# B&R Automation Studio project NAELD004C00R10L518F00 (part 17)

#### Act_OptP1025Save.st
```iecst
ACTION Act_OptP1025Save:

	IF tyP1025McSetAIVComm.tyAIVComm.tyNumSvrPort.bRtCompl OR tyP1025McSetAIVComm.tyAIVComm.tyNumAllwClntPort.bRtCompl
		OR tyP1025McSetAIVComm.tyAIVComm.tyStringAllwClntIP.bRtCompl THEN

		fUIInRtStatHide(ADR(tyCommon.tySet.tyBtnSave.uiMaskRtStat));

		 tyP1025McSetAIVComm.tyAIVComm.tyNumSvrPort.bRtCompl		:= FALSE;
		 tyP1025McSetAIVComm.tyAIVComm.tyNumAllwClntPort.bRtCompl	:= FALSE;
	 	 tyP1025McSetAIVComm.tyAIVComm.tyStringAllwClntIP.bRtCompl	:= FALSE;

	END_IF

	IF tyCommon.tySet.tyBtnSave.bRtCompl = TRUE THEN

		IF usiSaveAIVCommStep = 0 THEN
			//Verify IP Address Valid
			IF tyP1025McSetAIVComm.tyAIVComm.tyStringAllwClntIP.sValue <> '' THEN

				IF fIPValid(tyP1025McSetAIVComm.tyAIVComm.tyStringAllwClntIP.sValue, ADR(a_iIPPart1)) = TRUE THEN
					usiSaveAIVCommStep	:= 1;
				ELSE
					usiSaveAIVCommStep	:= 99;
				END_IF

			ELSE
				usiSaveAIVCommStep	:= 1;
			END_IF

		ELSIF usiSaveAIVCommStep = 1 THEN
			//Save Param
			tyMcParamWr.tyAIVComm.uiSvrPort			:=  DINT_TO_UINT(tyP1025McSetAIVComm.tyAIVComm.tyNumSvrPort.diValue);
			tyMcParamWr.tyAIVComm.uiClientPort		:=  DINT_TO_UINT(tyP1025McSetAIVComm.tyAIVComm.tyNumAllwClntPort.diValue);
			tyMcParamWr.tyAIVComm.sClientAddress	:=  tyP1025McSetAIVComm.tyAIVComm.tyStringAllwClntIP.sValue;

			eMcParamAct	:= McParamActWrite;

			IF p_eMcParamStat = McParamActWrite AND p_eMcParamStatus = Done THEN

				eMcParamAct	:= McParamActIdle;

				//Update BackUp Param
				tyP1025McSetAIVComm.tyAIVCommBkUp	:= tyP1025McSetAIVComm.tyAIVComm;

				//Reconnect
				bAIVCommReconnect	:= TRUE;

				usiSaveAIVCommStep	:= 2;

			ELSIF p_eMcParamStatus = Error THEN

				p_tyC0008MsgBox ACCESS ADR(tyP1025McSetAIVComm.tyMsgBoxSaveErr);

				IF tyP1025McSetAIVComm.tyMsgBoxSaveErr.tyBtnNo.bRtCompl = TRUE THEN
					tyP1025McSetAIVComm.tyMsgBoxSaveErr.tyBtnNo.bRtCompl	:= FALSE;
					tyP1025McSetAIVComm.tyMsgBoxSaveErr.tyBtnNo.bValue		:= FALSE;

					p_tyC0008MsgBox ACCESS ADR(tyP1025McSetAIVComm.tyMsgBoxHide);

					//Restore Param
					tyP1025McSetAIVComm.tyAIVComm	:= tyP1025McSetAIVComm.tyAIVCommBkUp;
					tyMcParamWr						:= p_tyMcParamCurr;

					tyCommon.tySet.tyBtnSave.bRtCompl	:= FALSE;
					fUIInRtStatOff(ADR(tyCommon.tySet.tyBtnSave.uiMaskRtStat));
				END_IF

			END_IF

		ELSIF usiSaveAIVCommStep = 2 THEN
			//Done
			bAIVCommReconnect	:= FALSE;

			usiSaveAIVCommStep	:= 0;

			tyCommon.tySet.tyBtnSave.bRtCompl 	:= FALSE;
			fUIInRtStatOff(ADR(tyCommon.tySet.tyBtnSave.uiMaskRtStat));

		ELSIF usiSaveAIVCommStep = 99 THEN
			//Message: IP Address Invalid
			p_tyC0008MsgBox ACCESS ADR(tyP1025McSetAIVComm.tyMsgBoxIPAddrInvalid);

			IF tyP1025McSetAIVComm.tyMsgBoxIPAddrInvalid.tyBtnNo.bRtCompl = TRUE THEN
				tyP1025McSetAIVComm.tyMsgBoxIPAddrInvalid.tyBtnNo.bRtCompl	:= FALSE;
				tyP1025McSetAIVComm.tyMsgBoxIPAddrInvalid.tyBtnNo.bValue	:= FALSE;

				p_tyC0008MsgBox ACCESS ADR(tyP1025McSetAIVComm.tyMsgBoxHide);

				//Restore Param
				tyP1025McSetAIVComm.tyAIVComm	:= tyP1025McSetAIVComm.tyAIVCommBkUp;

				usiSaveAIVCommStep	:= 0;

				tyCommon.tySet.tyBtnSave.bRtCompl	:= FALSE;
				fUIInRtStatOff(ADR(tyCommon.tySet.tyBtnSave.uiMaskRtStat));
			END_IF

		END_IF

	END_IF

END_ACTION
```

#### Act_EntP1026Disp.st
```iecst
ACTION Act_EntP1026Disp:

	//Access Address
	p_tyC0002FullMask ACCESS ADR(tyP1026McSetTeach.tyFullMaskHide);

	p_tyC0004Navi ACCESS ADR(tyP1026McSetTeach.tyNaviBack);

	p_tyC0005Main ACCESS ADR(tyCommon.tyMain);

	p_tyC0007Notif ACCESS ADR(tyCommon.tyNotif);

	p_tyC0008MsgBox ACCESS ADR(tyP1026McSetTeach.tyMsgBoxHide);

	p_tyC0009Info ACCESS ADR(tyCommon.tyInfo);

	p_tyP1026InOutletShutterFB ACCESS ADR(tyP1026McSetTeach.tyInOutletShutterFB);

	IF bTeachTravPosA = TRUE THEN
		p_tyP1026McSetTeach ACCESS ADR(tyP1026McSetTeach.tyTeachTravPosA);
		p_tyC0001MotionStd ACCESS ADR(tyP1026McSetTeach.tyMotionStdTrav);

	ELSIF bTeachTravPosB = TRUE THEN
		p_tyP1026McSetTeach ACCESS ADR(tyP1026McSetTeach.tyTeachTravPosB);
		p_tyC0001MotionStd ACCESS ADR(tyP1026McSetTeach.tyMotionStdTrav);

	ELSIF bTeachLifterPosA = TRUE THEN
		p_tyP1026McSetTeach ACCESS ADR(tyP1026McSetTeach.tyTeachLifterPosA);
		p_tyC0001MotionStd ACCESS ADR(tyP1026McSetTeach.tyMotionStdLifter);

	ELSIF bTeachLifterPosB = TRUE THEN
		p_tyP1026McSetTeach ACCESS ADR(tyP1026McSetTeach.tyTeachLifterPosB);
		p_tyC0001MotionStd ACCESS ADR(tyP1026McSetTeach.tyMotionStdLifter);

	END_IF

	//Display
	//Traverser
	tyP1026McSetTeach.tyMotionStdTrav.tyBtnPwr.bValue	:= p_bTravPwrOn;

	//Lifter
	tyP1026McSetTeach.tyMotionStdLifter.tyBtnPwr.bValue	:= p_bLifterBtmPwrOn;

//	bTeachServo		:= TRUE;
END_ACTION
```

#### Act_ExitP1026.st
```iecst
ACTION Act_ExitP1026:

	usiChgPage	:= 1;

	//Manual Deactivated
	bManualMod	:= FALSE;

	//Reset UI
	bJogSlow				:= FALSE;
	bJogFast				:= FALSE;
	fbJogSlowToFastDlyTm.IN	:= FALSE;

	fbLmtRstTm(IN := FALSE);
	//bypass curtain sensor
	bBypCurtainSen := FALSE;
	bBypCurtainPBLED := FALSE;
	tyP1026McSetTeach.tyTeachTravPosA.tyBtn4.bValue				:= FALSE;
	tyP1026McSetTeach.tyTeachTravPosB.tyBtn4.bValue				:= FALSE;
	tyP1026McSetTeach.tyTeachLifterPosA.tyBtn4.bValue				:= FALSE;
	tyP1026McSetTeach.tyTeachLifterPosB.tyBtn4.bValue				:= FALSE;

	//Traverser
	tyP1026McSetTeach.tyMotionStdTrav.tyBtnPwr.bRtCompl				:= FALSE;
	tyP1026McSetTeach.tyMotionStdTrav.tyBtnStop.bRtCompl			:= FALSE;
	tyP1026McSetTeach.tyMotionStdTrav.tyBtnOrigin.bRtCompl			:= FALSE;
	tyP1026McSetTeach.tyMotionStdTrav.tyBtnRst.bRtCompl				:= FALSE;
	tyP1026McSetTeach.tyMotionStdTrav.tyBtnMovAbs.bRtCompl			:= FALSE;
	tyP1026McSetTeach.tyMotionStdTrav.tyBtnMovRel.bRtCompl			:= FALSE;
	tyP1026McSetTeach.tyMotionStdTrav.tyBtnJogFront.bRtCompl		:= FALSE;
	tyP1026McSetTeach.tyMotionStdTrav.tyBtnJogRear.bRtCompl			:= FALSE;

	tyP1026McSetTeach.tyTeachTravPosA.tyBtn2.bRtCompl				:= FALSE;
	tyP1026McSetTeach.tyTeachTravPosB.tyBtn2.bRtCompl				:= FALSE;

	tyP1026McSetTeach.tyMotionStdTrav.tyBtnPwr.bValue				:= FALSE;
	tyP1026McSetTeach.tyMotionStdTrav.tyBtnStop.bValue				:= TRUE;
	tyP1026McSetTeach.tyMotionStdTrav.tyBtnOrigin.bValue			:= FALSE;
	tyP1026McSetTeach.tyMotionStdTrav.tyBtnRst.bValue				:= FALSE;
	tyP1026McSetTeach.tyMotionStdTrav.tyBtnMovAbs.bValue			:= FALSE;
	tyP1026McSetTeach.tyMotionStdTrav.tyBtnMovRel.bValue			:= FALSE;
	tyP1026McSetTeach.tyMotionStdTrav.tyBtnJogFront.bValue			:= FALSE;
	tyP1026McSetTeach.tyMotionStdTrav.tyBtnJogRear.bValue			:= FALSE;

	tyP1026McSetTeach.tyTeachTravPosA.tyBtn2.bValue					:= FALSE;
	tyP1026McSetTeach.tyTeachTravPosB.tyBtn2.bValue					:= FALSE;

	tyP1026McSetTeach.tyMotionStdTrav.tyBtnPwr.bRtLk				:= FALSE;
	tyP1026McSetTeach.tyMotionStdTrav.tyBtnStop.bRtLk				:= TRUE;
	tyP1026McSetTeach.tyMotionStdTrav.tyBtnOrigin.bRtLk				:= FALSE;
	tyP1026McSetTeach.tyMotionStdTrav.tyBtnRst.bRtLk				:= FALSE;
	tyP1026McSetTeach.tyMotionStdTrav.tyBtnMovAbs.bRtLk				:= FALSE;
	tyP1026McSetTeach.tyMotionStdTrav.tyBtnMovRel.bRtLk				:= FALSE;
	tyP1026McSetTeach.tyMotionStdTrav.tyBtnJogFront.bRtLk			:= FALSE;
	tyP1026McSetTeach.tyMotionStdTrav.tyBtnJogRear.bRtLk			:= FALSE;

	tyP1026McSetTeach.tyTeachTravPosA.tyBtn2.bRtLk					:= FALSE;
	tyP1026McSetTeach.tyTeachTravPosB.tyBtn2.bRtLk					:= FALSE;

	tyP1026McSetTeach.tyMotionStdTrav.tyBtnPwr.uiMaskRtStat			:= TRUE;
	tyP1026McSetTeach.tyMotionStdTrav.tyBtnOrigin.uiMaskRtStat		:= FALSE;
	tyP1026McSetTeach.tyMotionStdTrav.tyBtnRst.uiMaskRtStat			:= TRUE;
	tyP1026McSetTeach.tyMotionStdTrav.tyBtnMovAbs.uiMaskRtStat		:= FALSE;
	tyP1026McSetTeach.tyMotionStdTrav.tyBtnMovRel.uiMaskRtStat		:= FALSE;
	tyP1026McSetTeach.tyMotionStdTrav.tyBtnJogFront.uiMaskRtStat	:= FALSE;
	tyP1026McSetTeach.tyMotionStdTrav.tyBtnJogRear.uiMaskRtStat		:= FALSE;

	tyP1026McSetTeach.tyTeachTravPosA.tyBtn2.uiMaskRtStat			:= FALSE;
	tyP1026McSetTeach.tyTeachTravPosB.tyBtn2.uiMaskRtStat			:= FALSE;

	//Lifter
	tyP1026McSetTeach.tyMotionStdLifter.tyBtnPwr.bRtCompl			:= FALSE;
	tyP1026McSetTeach.tyMotionStdLifter.tyBtnStop.bRtCompl			:= FALSE;
	tyP1026McSetTeach.tyMotionStdLifter.tyBtnOrigin.bRtCompl		:= FALSE;
	tyP1026McSetTeach.tyMotionStdLifter.tyBtnRst.bRtCompl			:= FALSE;
	tyP1026McSetTeach.tyMotionStdLifter.tyBtnMovAbs.bRtCompl		:= FALSE;
	tyP1026McSetTeach.tyMotionStdLifter.tyBtnMovRel.bRtCompl		:= FALSE;
	tyP1026McSetTeach.tyMotionStdLifter.tyBtnJogUp.bRtCompl			:= FALSE;
	tyP1026McSetTeach.tyMotionStdLifter.tyBtnJogDown.bRtCompl		:= FALSE;

	tyP1026McSetTeach.tyTeachLifterPosA.tyBtn2.bRtCompl				:= FALSE;
	tyP1026McSetTeach.tyTeachLifterPosB.tyBtn2.bRtCompl				:= FALSE;

	tyP1026McSetTeach.tyMotionStdLifter.tyBtnPwr.bValue				:= FALSE;
	tyP1026McSetTeach.tyMotionStdLifter.tyBtnStop.bValue			:= TRUE;
	tyP1026McSetTeach.tyMotionStdLifter.tyBtnOrigin.bValue			:= FALSE;
	tyP1026McSetTeach.tyMotionStdLifter.tyBtnRst.bValue				:= FALSE;
	tyP1026McSetTeach.tyMotionStdLifter.tyBtnMovAbs.bValue			:= FALSE;
	tyP1026McSetTeach.tyMotionStdLifter.tyBtnMovRel.bValue			:= FALSE;
	tyP1026McSetTeach.tyMotionStdLifter.tyBtnJogUp.bValue			:= FALSE;
	tyP1026McSetTeach.tyMotionStdLifter.tyBtnJogDown.bValue			:= FALSE;

	tyP1026McSetTeach.tyTeachLifterPosA.tyBtn2.bValue				:= FALSE;
	tyP1026McSetTeach.tyTeachLifterPosB.tyBtn2.bValue				:= FALSE;

	tyP1026McSetTeach.tyMotionStdLifter.tyBtnPwr.bRtLk				:= FALSE;
	tyP1026McSetTeach.tyMotionStdLifter.tyBtnStop.bRtLk				:= TRUE;
	tyP1026McSetTeach.tyMotionStdLifter.tyBtnOrigin.bRtLk			:= FALSE;
	tyP1026McSetTeach.tyMotionStdLifter.tyBtnRst.bRtLk				:= FALSE;
	tyP1026McSetTeach.tyMotionStdLifter.tyBtnMovAbs.bRtLk			:= FALSE;
	tyP1026McSetTeach.tyMotionStdLifter.tyBtnMovRel.bRtLk			:= FALSE;
	tyP1026McSetTeach.tyMotionStdLifter.tyBtnJogUp.bRtLk			:= FALSE;
	tyP1026McSetTeach.tyMotionStdLifter.tyBtnJogDown.bRtLk			:= FALSE;

	tyP1026McSetTeach.tyTeachLifterPosA.tyBtn2.bRtLk				:= FALSE;
	tyP1026McSetTeach.tyTeachLifterPosB.tyBtn2.bRtLk				:= FALSE;

	tyP1026McSetTeach.tyMotionStdLifter.tyBtnPwr.uiMaskRtStat		:= TRUE;
	tyP1026McSetTeach.tyMotionStdLifter.tyBtnOrigin.uiMaskRtStat	:= FALSE;
	tyP1026McSetTeach.tyMotionStdLifter.tyBtnRst.uiMaskRtStat		:= TRUE;
	tyP1026McSetTeach.tyMotionStdLifter.tyBtnMovAbs.uiMaskRtStat	:= FALSE;
	tyP1026McSetTeach.tyMotionStdLifter.tyBtnMovRel.uiMaskRtStat	:= FALSE;
	tyP1026McSetTeach.tyMotionStdLifter.tyBtnJogUp.uiMaskRtStat		:= FALSE;
	tyP1026McSetTeach.tyMotionStdLifter.tyBtnJogDown.uiMaskRtStat	:= FALSE;

	tyP1026McSetTeach.tyTeachLifterPosA.tyBtn2.uiMaskRtStat			:= FALSE;
	tyP1026McSetTeach.tyTeachLifterPosB.tyBtn2.uiMaskRtStat			:= FALSE;

END_ACTION
```

#### Act_OptP1026TravTeach.st
```iecst
ACTION Act_OptP1026TravTeach:

	IF tyP1026McSetTeach.tyTeachTravPosA.tyBtn1.bRtCompl = TRUE THEN

		p_tyC0008MsgBox ACCESS ADR(tyP1026McSetTeach.tyMsgBoxUpdtTravPosA);

		IF tyP1026McSetTeach.tyMsgBoxUpdtTravPosA.tyBtnNo.bRtCompl THEN
			tyP1026McSetTeach.tyMsgBoxUpdtTravPosA.tyBtnNo.bRtCompl	:= FALSE;
			tyP1026McSetTeach.tyMsgBoxUpdtTravPosA.tyBtnNo.bValue	:= FALSE;

			p_tyC0008MsgBox ACCESS ADR(tyP1026McSetTeach.tyMsgBoxHide);

			//Write Actual Position To Machine Settings
			tyP1021McSetGen.tyGen.tyNumTravPosLaneA.diValue 	:= p_diTravActualPos;
			tyP1021McSetGen.tyGen.tyNumTravPosLaneA.bRtCompl	:= TRUE;

			//Back To Machine Settings
			eChgPage	:= UIP1021McSetGen;

			fUIInRtStatHide(ADR(tyCommon.tySet.tyBtnSave.uiMaskRtStat));

			tyP1026McSetTeach.tyTeachTravPosA.tyBtn1.bRtCompl	:= FALSE;
			tyP1026McSetTeach.tyTeachTravPosA.tyBtn1.bValue		:= FALSE;

		END_IF

	ELSIF tyP1026McSetTeach.tyTeachTravPosB.tyBtn1.bRtCompl = TRUE THEN

		p_tyC0008MsgBox ACCESS ADR(tyP1026McSetTeach.tyMsgBoxUpdtTravPosB);

		IF tyP1026McSetTeach.tyMsgBoxUpdtTravPosB.tyBtnNo.bRtCompl THEN
			tyP1026McSetTeach.tyMsgBoxUpdtTravPosB.tyBtnNo.bRtCompl := FALSE;
			tyP1026McSetTeach.tyMsgBoxUpdtTravPosB.tyBtnNo.bValue 	:= FALSE;

			p_tyC0008MsgBox ACCESS ADR(tyP1026McSetTeach.tyMsgBoxHide);

			//Write Actual Position To Machine Settings
			tyP1021McSetGen.tyGen.tyNumTravPosLaneB.diValue 	:= p_diTravActualPos;
			tyP1021McSetGen.tyGen.tyNumTravPosLaneB.bRtCompl	:= TRUE;

			//Back To Machine Settings
			eChgPage	:= UIP1021McSetGen;

			fUIInRtStatHide(ADR(tyCommon.tySet.tyBtnSave.uiMaskRtStat));

			tyP1026McSetTeach.tyTeachTravPosB.tyBtn1.bRtCompl	:= FALSE;
			tyP1026McSetTeach.tyTeachTravPosB.tyBtn1.bValue		:= FALSE;

		END_IF

	END_IF

END_ACTION
```

#### Act_OptP1026TravFBCtrl.st
```iecst
ACTION Act_OptP1026TravFBCtrl:

	fbJogSlowToFastDlyTm.PT			:= T#2s;
	fbJogSlowToFastDlyTm;
	fbLmtRstTm;

//	IF EDGEPOS((p_udiTravAxisErrID = 21570 OR p_udiTravAxisErrID = 21571)
	IF EDGEPOS((p_bTravFwdLmtSen OR p_bTravRevLmtSen OR p_udiTravAxisErrID = 21570 OR p_udiTravAxisErrID = 21571)
		AND tyP1026McSetTeach.tyMotionStdTrav.tyBtnJogRear.bValue = FALSE
		AND tyP1026McSetTeach.tyMotionStdTrav.tyBtnJogFront.bValue = FALSE) THEN

		fbLmtRstTm.IN				:= TRUE;
	END_IF

	IF fbLmtRstTm.Q = TRUE THEN
		tyP1026McSetTeach.tyMotionStdTrav.tyBtnRst.bRtCompl		:= TRUE;
	END_IF

	IF (tyP1026McSetTeach.tyMotionStdTrav.tyBtnJogFront.bValue = FALSE AND tyP1026McSetTeach.tyMotionStdTrav.tyBtnJogRear.bValue = FALSE) AND (p_bTravJogging = TRUE) THEN
		bJogStopTrav	:= TRUE;
	END_IF

	IF tyP1026McSetTeach.tyMotionStdTrav.tyBtnStop.bRtCompl = TRUE THEN
		eTravAct		:= TravActStop;

		IF p_eTravStat = TravActStop AND p_eTravStatus = Done THEN
			eTravAct	:= TravActIdle;

			tyP1026McSetTeach.tyMotionStdTrav.tyBtnStop.bRtCompl		:= FALSE;
			tyP1026McSetTeach.tyMotionStdTrav.tyBtnJogRear.bRtCompl		:= FALSE;
			tyP1026McSetTeach.tyMotionStdTrav.tyBtnJogFront.bRtCompl	:= FALSE;
			tyP1026McSetTeach.tyMotionStdTrav.tyBtnOrigin.bRtCompl		:= FALSE;
			tyP1026McSetTeach.tyMotionStdTrav.tyBtnMovAbs.bRtCompl		:= FALSE;
			tyP1026McSetTeach.tyMotionStdTrav.tyBtnMovRel.bRtCompl		:= FALSE;

			tyP1026McSetTeach.tyTeachTravPosA.tyBtn2.bRtCompl			:= FALSE;
			tyP1026McSetTeach.tyTeachTravPosB.tyBtn2.bRtCompl			:= FALSE;

			tyP1026McSetTeach.tyMotionStdTrav.tyBtnStop.bValue			:= TRUE;
			tyP1026McSetTeach.tyMotionStdTrav.tyBtnJogRear.bValue		:= FALSE;
			tyP1026McSetTeach.tyMotionStdTrav.tyBtnJogFront.bValue		:= FALSE;
			tyP1026McSetTeach.tyMotionStdTrav.tyBtnOrigin.bValue		:= FALSE;
			tyP1026McSetTeach.tyMotionStdTrav.tyBtnMovAbs.bValue		:= FALSE;
			tyP1026McSetTeach.tyMotionStdTrav.tyBtnMovRel.bValue		:= FALSE;
			tyP1026McSetTeach.tyTeachTravPosA.tyBtn2.bValue				:= FALSE;
			tyP1026McSetTeach.tyTeachTravPosB.tyBtn2.bValue				:= FALSE;

			tyP1026McSetTeach.tyMotionStdTrav.tyBtnStop.bRtLk			:= TRUE;
			tyP1026McSetTeach.tyMotionStdTrav.tyBtnJogRear.bRtLk		:= FALSE;
			tyP1026McSetTeach.tyMotionStdTrav.tyBtnJogFront.bRtLk		:= FALSE;
			tyP1026McSetTeach.tyMotionStdTrav.tyBtnOrigin.bRtLk			:= FALSE;
			tyP1026McSetTeach.tyMotionStdTrav.tyBtnMovAbs.bRtLk			:= FALSE;
			tyP1026McSetTeach.tyMotionStdTrav.tyBtnMovRel.bRtLk			:= FALSE;

			tyP1026McSetTeach.tyTeachTravPosA.tyBtn2.bRtLk						:= FALSE;
			tyP1026McSetTeach.tyTeachTravPosB.tyBtn2.bRtLk						:= FALSE;
		END_IF

	ELSIF (tyP1026McSetTeach.tyMotionStdTrav.tyBtnJogRear.bRtCompl = TRUE) OR (tyP1026McSetTeach.tyMotionStdTrav.tyBtnJogFront.bRtCompl = TRUE) OR (bJogStopTrav = TRUE) THEN
		bJogSlow					:= FALSE;
		bJogFast					:= FALSE;
		fbJogSlowToFastDlyTm.IN		:= FALSE;

		eTravAct		:= TravActJogStop;

		IF p_eTravStat = TravActJogStop AND p_eTravStatus = Done THEN
			eTravAct		:= TravActIdle;

			bJogStopTrav	:= FALSE;

			tyP1026McSetTeach.tyMotionStdTrav.tyBtnStop.bRtCompl		:= FALSE;
			tyP1026McSetTeach.tyMotionStdTrav.tyBtnJogRear.bRtCompl		:= FALSE;
			tyP1026McSetTeach.tyMotionStdTrav.tyBtnJogFront.bRtCompl	:= FALSE;
			tyP1026McSetTeach.tyMotionStdTrav.tyBtnOrigin.bRtCompl		:= FALSE;
			tyP1026McSetTeach.tyMotionStdTrav.tyBtnMovAbs.bRtCompl		:= FALSE;
			tyP1026McSetTeach.tyMotionStdTrav.tyBtnMovRel.bRtCompl		:= FALSE;
			tyP1026McSetTeach.tyTeachTravPosA.tyBtn2.bRtCompl			:= FALSE;
			tyP1026McSetTeach.tyTeachTravPosB.tyBtn2.bRtCompl			:= FALSE;

			tyP1026McSetTeach.tyMotionStdTrav.tyBtnStop.bValue			:= TRUE;
			tyP1026McSetTeach.tyMotionStdTrav.tyBtnJogRear.bValue		:= FALSE;
			tyP1026McSetTeach.tyMotionStdTrav.tyBtnJogFront.bValue		:= FALSE;
			tyP1026McSetTeach.tyMotionStdTrav.tyBtnOrigin.bValue		:= FALSE;
			tyP1026McSetTeach.tyMotionStdTrav.tyBtnMovAbs.bValue		:= FALSE;
			tyP1026McSetTeach.tyMotionStdTrav.tyBtnMovRel.bValue		:= FALSE;
			tyP1026McSetTeach.tyTeachTravPosA.tyBtn2.bValue				:= FALSE;
			tyP1026McSetTeach.tyTeachTravPosB.tyBtn2.bValue				:= FALSE;

			tyP1026McSetTeach.tyMotionStdTrav.tyBtnStop.bRtLk			:= TRUE;
			tyP1026McSetTeach.tyMotionStdTrav.tyBtnJogRear.bRtLk		:= FALSE;
			tyP1026McSetTeach.tyMotionStdTrav.tyBtnJogFront.bRtLk		:= FALSE;
			tyP1026McSetTeach.tyMotionStdTrav.tyBtnOrigin.bRtLk			:= FALSE;
			tyP1026McSetTeach.tyMotionStdTrav.tyBtnMovAbs.bRtLk			:= FALSE;
			tyP1026McSetTeach.tyMotionStdTrav.tyBtnMovRel.bRtLk			:= FALSE;
			tyP1026McSetTeach.tyTeachTravPosA.tyBtn2.bRtLk				:= FALSE;
			tyP1026McSetTeach.tyTeachTravPosB.tyBtn2.bRtLk				:= FALSE;
		END_IF

	ELSIF tyP1026McSetTeach.tyMotionStdTrav.tyBtnPwr.bRtCompl = TRUE THEN
		tyP1026McSetTeach.tyMotionStdTrav.tyBtnPwr.bRtLk				:= TRUE;

		IF tyP1026McSetTeach.tyMotionStdTrav.tyBtnPwr.bValue = TRUE THEN
			eTravAct		:= TravActPwrOn;

			IF p_eTravStat = TravActPwrOn AND p_eTravStatus = Done THEN
				eTravAct	:= TravActIdle;

				tyP1026McSetTeach.tyMotionStdTrav.tyBtnPwr.bRtCompl		:= FALSE;
				tyP1026McSetTeach.tyMotionStdTrav.tyBtnPwr.bRtLk		:= FALSE;
			END_IF
		ELSE
			eTravAct		:= TravActPwrOff;

			IF p_eTravStat = TravActPwrOff AND p_eTravStatus = Done THEN
				eTravAct	:= TravActIdle;

				tyP1026McSetTeach.tyMotionStdTrav.tyBtnPwr.bRtCompl		:= FALSE;
				tyP1026McSetTeach.tyMotionStdTrav.tyBtnPwr.bRtLk		:= FALSE;
			END_IF
		END_IF

	ELSIF tyP1026McSetTeach.tyMotionStdTrav.tyBtnOrigin.bRtCompl = TRUE THEN
		tyP1026McSetTeach.tyMotionStdTrav.tyBtnOrigin.bValue			:= TRUE;
		tyP1026McSetTeach.tyMotionStdTrav.tyBtnStop.bValue				:= FALSE;

		tyP1026McSetTeach.tyMotionStdTrav.tyBtnOrigin.bRtLk				:= TRUE;
		tyP1026McSetTeach.tyMotionStdTrav.tyBtnStop.bRtLk				:= FALSE;

		eTravAct		:= TravActHoming;

		IF p_eTravStat = TravActHoming AND p_eTravStatus = Done THEN
			eTravAct	:= TravActIdle;

			tyP1026McSetTeach.tyMotionStdTrav.tyBtnOrigin.bRtCompl		:= FALSE;
			tyP1026McSetTeach.tyMotionStdTrav.tyBtnOrigin.bValue		:= FALSE;
			tyP1026McSetTeach.tyMotionStdTrav.tyBtnStop.bValue			:= TRUE;

			tyP1026McSetTeach.tyMotionStdTrav.tyBtnOrigin.bRtLk			:= FALSE;
			tyP1026McSetTeach.tyMotionStdTrav.tyBtnStop.bRtLk			:= TRUE;
		END_IF

	ELSIF tyP1026McSetTeach.tyMotionStdTrav.tyBtnRst.bRtCompl = TRUE THEN
		tyP1026McSetTeach.tyMotionStdTrav.tyBtnRst.bValue				:= TRUE;
		tyP1026McSetTeach.tyMotionStdTrav.tyBtnRst.bRtLk				:= TRUE;

		eTravAct		:= TravActRstAxisErr;

		IF p_eTravStat = TravActRstAxisErr AND p_eTravStatus = Done THEN
			eTravAct	:= TravActIdle;

			tyP1026McSetTeach.tyMotionStdTrav.tyBtnRst.bRtCompl			:= FALSE;
			tyP1026McSetTeach.tyMotionStdTrav.tyBtnRst.bValue			:= FALSE;
			tyP1026McSetTeach.tyMotionStdTrav.tyBtnRst.bRtLk			:= FALSE;

			fbLmtRstTm.IN			:= FALSE;
		END_IF

	ELSIF tyP1026McSetTeach.tyTeachTravPosA.tyBtn2.bRtCompl = TRUE THEN
		tyP1026McSetTeach.tyTeachTravPosA.tyBtn2.bValue		:= TRUE;
		tyP1026McSetTeach.tyMotionStdTrav.tyBtnStop.bValue	:= FALSE;

		tyP1026McSetTeach.tyTeachTravPosA.tyBtn2.bRtLk		:= TRUE;
		tyP1026McSetTeach.tyMotionStdTrav.tyBtnStop.bRtLk	:= FALSE;

		diMnlTravNomSpd	:= tyP1026McSetTeach.tyMotionStdTrav.tyNumNomSpd.diValue;

		eTravAct		:= TravActGoDPos;

		IF p_eTravStat = TravActGoDPos AND p_eTravStatus = Done THEN
			eTravAct	:= TravActIdle;

			tyP1026McSetTeach.tyTeachTravPosA.tyBtn2.bRtCompl	:= FALSE;
			tyP1026McSetTeach.tyTeachTravPosA.tyBtn2.bValue		:= FALSE;
			tyP1026McSetTeach.tyMotionStdTrav.tyBtnStop.bValue	:= TRUE;

			tyP1026McSetTeach.tyTeachTravPosA.tyBtn2.bRtLk		:= FALSE;
			tyP1026McSetTeach.tyMotionStdTrav.tyBtnStop.bRtLk	:= TRUE;
		END_IF

	ELSIF tyP1026McSetTeach.tyTeachTravPosB.tyBtn2.bRtCompl = TRUE THEN
		tyP1026McSetTeach.tyTeachTravPosB.tyBtn2.bValue		:= TRUE;
		tyP1026McSetTeach.tyMotionStdTrav.tyBtnStop.bValue	:= FALSE;

		tyP1026McSetTeach.tyTeachTravPosB.tyBtn2.bRtLk		:= TRUE;
		tyP1026McSetTeach.tyMotionStdTrav.tyBtnStop.bRtLk	:= FALSE;

		diMnlTravNomSpd	:= tyP1026McSetTeach.tyMotionStdTrav.tyNumNomSpd.diValue;

		eTravAct		:= TravActGoEPos;

		IF p_eTravStat = TravActGoEPos AND p_eTravStatus = Done THEN
			eTravAct	:= TravActIdle;

			tyP1026McSetTeach.tyTeachTravPosB.tyBtn2.bRtCompl	:= FALSE;
			tyP1026McSetTeach.tyTeachTravPosB.tyBtn2.bValue		:= FALSE;
			tyP1026McSetTeach.tyMotionStdTrav.tyBtnStop.bValue	:= TRUE;

			tyP1026McSetTeach.tyTeachTravPosB.tyBtn2.bRtLk		:= FALSE;
			tyP1026McSetTeach.tyMotionStdTrav.tyBtnStop.bRtLk	:= TRUE;
		END_IF

	ELSIF tyP1026McSetTeach.tyMotionStdTrav.tyBtnMovAbs.bRtCompl = TRUE THEN
		tyP1026McSetTeach.tyMotionStdTrav.tyBtnMovAbs.bValue	:= TRUE;
		tyP1026McSetTeach.tyMotionStdTrav.tyBtnStop.bValue		:= FALSE;

		tyP1026McSetTeach.tyMotionStdTrav.tyBtnMovAbs.bRtLk		:= TRUE;
		tyP1026McSetTeach.tyMotionStdTrav.tyBtnStop.bRtLk		:= FALSE;

		diMnlTravTargetPos	:= tyP1026McSetTeach.tyMotionStdTrav.tyNumTargetPos.diValue;
		diMnlTravNomSpd		:= tyP1026McSetTeach.tyMotionStdTrav.tyNumNomSpd.diValue;

		eTravAct		:= TravActMovAbs;

		IF p_eTravStat = TravActMovAbs AND p_eTravStatus = Done THEN
			eTravAct	:= TravActIdle;

			tyP1026McSetTeach.tyMotionStdTrav.tyBtnMovAbs.bRtCompl		:= FALSE;
			tyP1026McSetTeach.tyMotionStdTrav.tyBtnMovAbs.bValue		:= FALSE;
			tyP1026McSetTeach.tyMotionStdTrav.tyBtnStop.bValue			:= TRUE;

			tyP1026McSetTeach.tyMotionStdTrav.tyBtnMovAbs.bRtLk			:= FALSE;
			tyP1026McSetTeach.tyMotionStdTrav.tyBtnStop.bRtLk			:= TRUE;
		END_IF

	ELSIF tyP1026McSetTeach.tyMotionStdTrav.tyBtnMovRel.bRtCompl = TRUE THEN
		tyP1026McSetTeach.tyMotionStdTrav.tyBtnMovRel.bValue			:= TRUE;
		tyP1026McSetTeach.tyMotionStdTrav.tyBtnStop.bValue				:= FALSE;

		tyP1026McSetTeach.tyMotionStdTrav.tyBtnMovRel.bRtLk				:= TRUE;
		tyP1026McSetTeach.tyMotionStdTrav.tyBtnStop.bRtLk				:= FALSE;

		diMnlTravStepSize	:= tyP1026McSetTeach.tyMotionStdTrav.tyNumStepSize.diValue;
		diMnlTravNomSpd		:= tyP1026McSetTeach.tyMotionStdTrav.tyNumNomSpd.diValue;

		eTravAct		:= TravActMovRel;

		IF p_eTravStat = TravActMovRel AND p_eTravStatus = Done THEN
			eTravAct	:= TravActIdle;

			tyP1026McSetTeach.tyMotionStdTrav.tyBtnMovRel.bRtCompl		:= FALSE;
			tyP1026McSetTeach.tyMotionStdTrav.tyBtnMovRel.bValue		:= FALSE;
			tyP1026McSetTeach.tyMotionStdTrav.tyBtnStop.bValue			:= TRUE;

			tyP1026McSetTeach.tyMotionStdTrav.tyBtnMovRel.bRtLk			:= FALSE;
			tyP1026McSetTeach.tyMotionStdTrav.tyBtnStop.bRtLk			:= TRUE;
		END_IF

	ELSIF (tyP1026McSetTeach.tyMotionStdTrav.tyBtnJogRear.bValue = TRUE) AND (fbJogSlowToFastDlyTm.Q = FALSE) AND (bJogSlow = FALSE) THEN
		tyP1026McSetTeach.tyMotionStdTrav.tyBtnStop.bValue				:= FALSE;
		tyP1026McSetTeach.tyMotionStdTrav.tyBtnStop.bRtLk				:= FALSE;

		fbJogSlowToFastDlyTm.IN		:= TRUE;

		diMnlTravJogSpd	:= tyP1026McSetTeach.tyMotionStdTrav.tyNumSlwSpd.diValue;

		eTravAct		:= TravActJogRear;

		IF p_eTravStat = TravActJogRear AND p_eTravStatus = Done THEN
			eTravAct	:= TravActIdle;
			bJogSlow				:= TRUE;
		ELSIF p_eTravStatus = Error THEN
			fbJogSlowToFastDlyTm.IN	:= FALSE;
			bJogSlow				:= TRUE;
		END_IF

	ELSIF (tyP1026McSetTeach.tyMotionStdTrav.tyBtnJogRear.bValue = TRUE) AND (fbJogSlowToFastDlyTm.Q = TRUE) AND (bJogFast = FALSE) THEN
		tyP1026McSetTeach.tyMotionStdTrav.tyBtnStop.bValue					:= FALSE;
		tyP1026McSetTeach.tyMotionStdTrav.tyBtnStop.bRtLk					:= FALSE;

		fbJogSlowToFastDlyTm.IN		:= TRUE;

		diMnlTravJogSpd	:= tyP1026McSetTeach.tyMotionStdTrav.tyNumNomSpd.diValue;

		eTravAct		:= TravActJogRear;

		IF p_eTravStat = TravActJogRear AND p_eTravStatus = Done THEN
			eTravAct	:= TravActIdle;
			bJogFast				:= TRUE;
		ELSIF p_eTravStatus = Error THEN
			fbJogSlowToFastDlyTm.IN	:= FALSE;
			bJogFast				:= TRUE;
		END_IF

	ELSIF (tyP1026McSetTeach.tyMotionStdTrav.tyBtnJogFront.bValue = TRUE) AND (fbJogSlowToFastDlyTm.Q = FALSE) AND (bJogSlow = FALSE) THEN
		tyP1026McSetTeach.tyMotionStdTrav.tyBtnStop.bValue				:= FALSE;
		tyP1026McSetTeach.tyMotionStdTrav.tyBtnStop.bRtLk				:= FALSE;

		fbJogSlowToFastDlyTm.IN		:= TRUE;

		diMnlTravJogSpd	:= tyP1026McSetTeach.tyMotionStdTrav.tyNumSlwSpd.diValue;

		eTravAct		:= TravActJogFront;

		IF p_eTravStat = TravActJogFront AND p_eTravStatus = Done THEN
			eTravAct	:= TravActIdle;
			bJogSlow				:= TRUE;
		ELSIF p_eTravStatus = Error THEN
			fbJogSlowToFastDlyTm.IN	:= FALSE;
			bJogSlow				:= TRUE;
		END_IF

	ELSIF (tyP1026McSetTeach.tyMotionStdTrav.tyBtnJogFront.bValue = TRUE) AND (fbJogSlowToFastDlyTm.Q = TRUE) AND (bJogFast = FALSE) THEN
		tyP1026McSetTeach.tyMotionStdTrav.tyBtnStop.bValue				:= FALSE;
		tyP1026McSetTeach.tyMotionStdTrav.tyBtnStop.bRtLk				:= FALSE;

		fbJogSlowToFastDlyTm.IN		:= TRUE;

		diMnlTravJogSpd	:= tyP1026McSetTeach.tyMotionStdTrav.tyNumNomSpd.diValue;

		eTravAct	:= TravActJogFront;

		IF p_eTravStat = TravActJogFront AND p_eTravStatus = Done THEN
			eTravAct	:= TravActIdle;
			bJogFast	:= TRUE;
		ELSIF p_eTravStatus = Error THEN
			fbJogSlowToFastDlyTm.IN	:= FALSE;
			bJogFast				:= TRUE;
		END_IF

	END_IF

	IF tyP1026McSetTeach.tyInOutletShutterFB.tyBtnOpen.bRtCompl = TRUE THEN
		tyP1026McSetTeach.tyInOutletShutterFB.tyBtnOpen.bRtCompl	:= FALSE;

		tyP1026McSetTeach.tyInOutletShutterFB.tyBtnOpen.bValue	:= TRUE;
		tyP1026McSetTeach.tyInOutletShutterFB.tyBtnClose.bValue	:= FALSE;

	ELSIF tyP1026McSetTeach.tyInOutletShutterFB.tyBtnClose.bRtCompl = TRUE THEN
		tyP1026McSetTeach.tyInOutletShutterFB.tyBtnClose.bRtCompl	:= FALSE;

		tyP1026McSetTeach.tyInOutletShutterFB.tyBtnClose.bValue	:= TRUE;
		tyP1026McSetTeach.tyInOutletShutterFB.tyBtnOpen.bValue	:= FALSE;
	END_IF

	IF tyP1026McSetTeach.tyInOutletShutterFB.tyBtnOpen.bValue = TRUE THEN
		eInShutterAct	:= PneuActRet;
		eInShutterAct2	:= PneuActRet;
		eInShutterAct3	:= PneuActRet;
		eOutShutterAct	:= PneuActRet;

		IF (p_eInShutterStat = PneuActRet AND p_eInShutterStatus = Done)
			AND (p_eOutShutterStat = PneuActRet AND p_eOutShutterStatus = Done)
			THEN
			eInShutterAct	:= PneuActIdle;
			eInShutterAct2	:= PneuActIdle;
			eInShutterAct3	:= PneuActIdle;
			eOutShutterAct	:= PneuActIdle;
			tyP1026McSetTeach.tyInOutletShutterFB.tyBtnOpen.bValue	:= FALSE;
		ELSIF p_eInShutterStatus = Error OR p_eOutShutterStatus = Error THEN
			tyP1026McSetTeach.tyInOutletShutterFB.tyBtnOpen.bValue	:= FALSE;
		END_IF

	ELSIF tyP1026McSetTeach.tyInOutletShutterFB.tyBtnClose.bValue = TRUE THEN
		eInShutterAct	:= PneuActExt;
		eInShutterAct2	:= PneuActExt;
		eInShutterAct3	:= PneuActExt;
		eOutShutterAct	:= PneuActExt;
		IF (p_eInShutterStat = PneuActExt AND p_eInShutterStatus = Done)
			AND (p_eOutShutterStat = PneuActExt AND p_eOutShutterStatus = Done)
			THEN
			eInShutterAct	:= PneuActIdle;
			eInShutterAct2	:= PneuActIdle;
			eInShutterAct3	:= PneuActIdle;
			eOutShutterAct	:= PneuActIdle;
			tyP1026McSetTeach.tyInOutletShutterFB.tyBtnClose.bValue := FALSE;
		ELSIF p_eInShutterStatus = Error OR p_eOutShutterStatus = Error THEN
			tyP1026McSetTeach.tyInOutletShutterFB.tyBtnClose.bValue := FALSE;
		END_IF
	END_IF

	//bypass curtain sensor
	IF bTeachTravPosA OR bTeachTravPosB THEN
		bBypCurtainSen			:= tyP1026McSetTeach.tyTeachTravPosA.tyBtn4.bValue OR tyP1026McSetTeach.tyTeachTravPosB.tyBtn4.bValue;
		bBypCurtainPBLED		:= tyP1026McSetTeach.tyTeachTravPosA.tyBtn4.bValue OR tyP1026McSetTeach.tyTeachTravPosB.tyBtn4.bValue;
	END_IF

END_ACTION
```

#### Act_OptP1026TravUpdtDat.st
```iecst
ACTION Act_OptP1026TravUpdtDat:

	tyP1026McSetTeach.tyMotionStdTrav.tyNumCurrPos.diValue			:= p_diTravActualPos;
	tyP1026McSetTeach.tyMotionStdTrav.tyNumErrCode.diValue			:= UDINT_TO_DINT(p_udiTravAxisErrID);
	tyP1026McSetTeach.tyMotionStdTrav.tyBitmapPwr.usiValueIdx		:= BOOL_TO_USINT(p_bTravPwrOn);
	tyP1026McSetTeach.tyMotionStdTrav.tyBitmapRst.usiValueIdx		:= BOOL_TO_USINT(NOT p_bTravAxisErr);
	tyP1026McSetTeach.tyMotionStdTrav.tyBitmapOrigin.usiValueIdx	:= BOOL_TO_USINT(p_bTravIsHomed);
	tyP1026McSetTeach.tyMotionStdTrav.tyBtnFrontLmtSen.bValue		:= p_bTravFrontSen;
	tyP1026McSetTeach.tyMotionStdTrav.tyBtnRearLmtSen.bValue		:= p_bTravRearSen;

	//Machine Bitmap
	IF   (p_tyNtParamCurr.eProjMag = LDMagDual AND p_tyNtParamCurr.bMagAutoVerifyPrep = FALSE)
		OR (p_tyNtParamCurr.eProjMag = LDMagTriple AND p_tyNtParamCurr.bMagAutoVerifyPrep = FALSE)
		OR (p_tyNtParamCurr.eProjMag = LDMagDual AND p_tyNtParamCurr.bMagAutoVerifyPrep = TRUE)
		THEN
		IF p_bTravIsHomed = TRUE THEN
			IF p_diTravActualPos <= (p_tyNtParamCurr.tyUITravTargetPos.diMax / 3) THEN
				tyP1026McSetTeach.tyMotionStdTrav.tyBitmapMc.uiValueIdx 	:= 5;
			ELSIF p_diTravActualPos <= (p_tyNtParamCurr.tyUITravTargetPos.diMax / 3 * 2) THEN
				tyP1026McSetTeach.tyMotionStdTrav.tyBitmapMc.uiValueIdx 	:= 6;
			ELSE
				tyP1026McSetTeach.tyMotionStdTrav.tyBitmapMc.uiValueIdx 	:= 7;
			END_IF
		ELSE
			tyP1026McSetTeach.tyMotionStdTrav.tyBitmapMc.uiValueIdx	:= 5;
		END_IF
	ELSIF p_tyNtParamCurr.eProjMag = LDMagTriple AND p_tyNtParamCurr.bMagAutoVerifyPrep = TRUE
		THEN
		IF p_bTravIsHomed = TRUE THEN
			IF p_diTravActualPos <= (p_tyNtParamCurr.tyUITravTargetPos.diMax / 3) THEN
				tyP1026McSetTeach.tyMotionStdTrav.tyBitmapMc.uiValueIdx 	:= 26;
			ELSIF p_diTravActualPos <= (p_tyNtParamCurr.tyUITravTargetPos.diMax / 3 * 2) THEN
				tyP1026McSetTeach.tyMotionStdTrav.tyBitmapMc.uiValueIdx 	:= 27;
			ELSE
				tyP1026McSetTeach.tyMotionStdTrav.tyBitmapMc.uiValueIdx 	:= 28;
			END_IF
		ELSE
			tyP1026McSetTeach.tyMotionStdTrav.tyBitmapMc.uiValueIdx	:= 26;
		END_IF
	ELSIF p_tyNtParamCurr.eProjMag = LDMagQuadruple AND p_tyNtParamCurr.bMagAutoVerifyPrep = TRUE
		THEN
		IF p_bTravIsHomed = TRUE THEN
			IF p_diTravActualPos <= (p_tyNtParamCurr.tyUITravTargetPos.diMax / 3) THEN
				tyP1026McSetTeach.tyMotionStdTrav.tyBitmapMc.uiValueIdx 	:= 45;
			ELSIF p_diTravActualPos <= (p_tyNtParamCurr.tyUITravTargetPos.diMax / 3 * 2) THEN
				tyP1026McSetTeach.tyMotionStdTrav.tyBitmapMc.uiValueIdx 	:= 46;
			ELSE
				tyP1026McSetTeach.tyMotionStdTrav.tyBitmapMc.uiValueIdx 	:= 47;
			END_IF
		ELSE
			tyP1026McSetTeach.tyMotionStdTrav.tyBitmapMc.uiValueIdx	:= 45;
		END_IF
	END_IF

	IF p_tyNtParamCurr.eProjMag = LDMagTriple AND p_tyNtParamCurr.bProjLifterMagPlatform THEN
		IF 	tyP1026McSetTeach.tyMotionStdTrav.tyBitmapMc.uiValueIdx < 400 THEN
			tyP1026McSetTeach.tyMotionStdTrav.tyBitmapMc.uiValueIdx	:= tyP1026McSetTeach.tyMotionStdTrav.tyBitmapMc.uiValueIdx + 400;
		END_IF
	ELSIF p_tyNtParamCurr.eProjMag = LDMagTriple AND p_tyNtParamCurr.bMagAutoVerifyPrep = FALSE AND p_tyNtParamCurr.bProjMotorizedPullerPrep = FALSE THEN
		IF 	tyP1026McSetTeach.tyMotionStdTrav.tyBitmapMc.uiValueIdx < 100 THEN
			tyP1026McSetTeach.tyMotionStdTrav.tyBitmapMc.uiValueIdx	:= tyP1026McSetTeach.tyMotionStdTrav.tyBitmapMc.uiValueIdx + 100;
		END_IF
	ELSIF p_tyNtParamCurr.eProjMag = LDMagDual AND p_tyNtParamCurr.bMagAutoVerifyPrep = FALSE THEN
		IF 	tyP1026McSetTeach.tyMotionStdTrav.tyBitmapMc.uiValueIdx < 100 THEN
			IF p_tyNtParamCurr.sJobNo = '2023-0258A01' THEN
				tyP1026McSetTeach.tyMotionStdTrav.tyBitmapMc.uiValueIdx	:= tyP1026McSetTeach.tyMotionStdTrav.tyBitmapMc.uiValueIdx + 447-5;
			ELSE
				tyP1026McSetTeach.tyMotionStdTrav.tyBitmapMc.uiValueIdx	:= tyP1026McSetTeach.tyMotionStdTrav.tyBitmapMc.uiValueIdx + 200;
			END_IF
		END_IF
	ELSIF (p_tyNtParamCurr.eProjMag = LDMagDual OR p_tyNtParamCurr.eProjMag = LDMagTriple)
		AND p_tyNtParamCurr.bMagAutoVerifyPrep = TRUE THEN
		IF 	tyP1026McSetTeach.tyMotionStdTrav.tyBitmapMc.uiValueIdx < 200 THEN
			tyP1026McSetTeach.tyMotionStdTrav.tyBitmapMc.uiValueIdx	:= tyP1026McSetTeach.tyMotionStdTrav.tyBitmapMc.uiValueIdx + 200;
		END_IF
	ELSIF p_tyNtParamCurr.eProjMag = LDMagTriple AND p_tyNtParamCurr.bMagAutoVerifyPrep = FALSE AND p_tyNtParamCurr.bProjMotorizedPullerPrep = TRUE THEN
		IF 	tyP1026McSetTeach.tyMotionStdTrav.tyBitmapMc.uiValueIdx < 300 THEN
			tyP1026McSetTeach.tyMotionStdTrav.tyBitmapMc.uiValueIdx	:= tyP1026McSetTeach.tyMotionStdTrav.tyBitmapMc.uiValueIdx + 300;
		END_IF
	END_IF

END_ACTION
```

#### Act_OptP1026LifterTeach.st
```iecst
ACTION Act_OptP1026LifterTeach:

	IF tyP1026McSetTeach.tyTeachLifterPosA.tyBtn1.bRtCompl = TRUE THEN

		p_tyC0008MsgBox ACCESS ADR(tyP1026McSetTeach.tyMsgBoxUpdtLifterPosA);

		IF tyP1026McSetTeach.tyMsgBoxUpdtLifterPosA.tyBtnNo.bRtCompl THEN
			tyP1026McSetTeach.tyMsgBoxUpdtLifterPosA.tyBtnNo.bRtCompl	:= FALSE;
			tyP1026McSetTeach.tyMsgBoxUpdtLifterPosA.tyBtnNo.bValue		:= FALSE;

			p_tyC0008MsgBox ACCESS ADR(tyP1026McSetTeach.tyMsgBoxHide);

			//Write Actual Position To Machine Settings
			tyP1021McSetGen.tyGen.tyNumLiftPosLaneA.diValue		:= p_diLifterBtmActualPos;
			tyP1021McSetGen.tyGen.tyNumLiftPosLaneA.bRtCompl	:= TRUE;

			//Back To Machine Settings
			eChgPage	:= UIP1021McSetGen;

			fUIInRtStatHide(ADR(tyCommon.tySet.tyBtnSave.uiMaskRtStat));

			tyP1026McSetTeach.tyTeachLifterPosA.tyBtn1.bRtCompl	:= FALSE;
			tyP1026McSetTeach.tyTeachLifterPosA.tyBtn1.bValue	:= FALSE;

		END_IF

	ELSIF tyP1026McSetTeach.tyTeachLifterPosB.tyBtn1.bRtCompl = TRUE THEN

		p_tyC0008MsgBox ACCESS ADR(tyP1026McSetTeach.tyMsgBoxUpdtLifterPosB);

		IF tyP1026McSetTeach.tyMsgBoxUpdtLifterPosB.tyBtnNo.bRtCompl THEN
			tyP1026McSetTeach.tyMsgBoxUpdtLifterPosB.tyBtnNo.bRtCompl	:= FALSE;
			tyP1026McSetTeach.tyMsgBoxUpdtLifterPosB.tyBtnNo.bValue		:= FALSE;

			p_tyC0008MsgBox ACCESS ADR(tyP1026McSetTeach.tyMsgBoxHide);

			//Write Actual Position To Machine Settings
			tyP1021McSetGen.tyGen.tyNumLiftPosLaneB.diValue		:= p_diLifterBtmActualPos;
			tyP1021McSetGen.tyGen.tyNumLiftPosLaneB.bRtCompl	:= TRUE;

			//Back To Machine Settings
			eChgPage	:= UIP1021McSetGen;

			fUIInRtStatHide(ADR(tyCommon.tySet.tyBtnSave.uiMaskRtStat));

			tyP1026McSetTeach.tyTeachLifterPosB.tyBtn1.bRtCompl	:= FALSE;
			tyP1026McSetTeach.tyTeachLifterPosB.tyBtn1.bValue	:= FALSE;

		END_IF

	END_IF

END_ACTION
```

#### Act_OptP1026LifterFBCtrl.st
```iecst
ACTION Act_OptP1026LifterFBCtrl:

	fbJogSlowToFastDlyTm.PT	:= T#2s;
	fbJogSlowToFastDlyTm;
	fbLmtRstTm;

	//Lifter Safety Sensor Interruption
	IF EDGENEG(p_tyDI.bLifterSafetyLmtSW1 AND p_tyDI.bLifterSafetyLmtSW2 AND p_tyDI.bLifterTimingBeltSen) THEN
		tyP1026McSetTeach.tyMotionStdLifter.tyBtnStop.bRtCompl	:= TRUE;
	END_IF

//	IF EDGEPOS((p_udiLifterBtmAxisErrID = 21570 OR p_udiLifterBtmAxisErrID = 21571)
	IF EDGEPOS((p_bLifterBtmFwdLmtSen OR p_bLifterBtmRevLmtSen OR p_udiLifterBtmAxisErrID = 21570 OR p_udiLifterBtmAxisErrID = 21571)
		AND tyP1026McSetTeach.tyMotionStdLifter.tyBtnJogDown.bValue = FALSE
		AND tyP1026McSetTeach.tyMotionStdLifter.tyBtnJogUp.bValue = FALSE) THEN
		fbLmtRstTm.IN	:= TRUE;
	END_IF

	IF fbLmtRstTm.Q = TRUE THEN
		tyP1026McSetTeach.tyMotionStdLifter.tyBtnRst.bRtCompl	:= TRUE;
	END_IF

	IF (tyP1026McSetTeach.tyMotionStdLifter.tyBtnJogUp.bValue = FALSE AND tyP1026McSetTeach.tyMotionStdLifter.tyBtnJogDown.bValue = FALSE) AND (p_bLifterBtmJogging = TRUE) THEN
		bJogStopLifter	:= TRUE;
	END_IF

	IF tyP1026McSetTeach.tyMotionStdLifter.tyBtnStop.bRtCompl = TRUE THEN
		eLifterBtmAct		:= LifterActStop;

		IF p_eLifterBtmStat = LifterActStop AND p_eLifterBtmStatus = Done THEN
			eLifterBtmAct	:= LifterActIdle;

			tyP1026McSetTeach.tyMotionStdLifter.tyBtnStop.bRtCompl			:= FALSE;
			tyP1026McSetTeach.tyMotionStdLifter.tyBtnJogDown.bRtCompl		:= FALSE;
			tyP1026McSetTeach.tyMotionStdLifter.tyBtnJogUp.bRtCompl			:= FALSE;
			tyP1026McSetTeach.tyMotionStdLifter.tyBtnOrigin.bRtCompl		:= FALSE;
			tyP1026McSetTeach.tyMotionStdLifter.tyBtnMovAbs.bRtCompl		:= FALSE;
			tyP1026McSetTeach.tyMotionStdLifter.tyBtnMovRel.bRtCompl		:= FALSE;

			tyP1026McSetTeach.tyTeachLifterPosA.tyBtn2.bRtCompl				:= FALSE;
			tyP1026McSetTeach.tyTeachLifterPosB.tyBtn2.bRtCompl				:= FALSE;

			tyP1026McSetTeach.tyMotionStdLifter.tyBtnStop.bValue			:= TRUE;
			tyP1026McSetTeach.tyMotionStdLifter.tyBtnJogDown.bValue			:= FALSE;
			tyP1026McSetTeach.tyMotionStdLifter.tyBtnJogUp.bValue			:= FALSE;
			tyP1026McSetTeach.tyMotionStdLifter.tyBtnOrigin.bValue			:= FALSE;
			tyP1026McSetTeach.tyMotionStdLifter.tyBtnMovAbs.bValue			:= FALSE;
			tyP1026McSetTeach.tyMotionStdLifter.tyBtnMovRel.bValue			:= FALSE;

			tyP1026McSetTeach.tyTeachLifterPosA.tyBtn2.bValue				:= FALSE;
			tyP1026McSetTeach.tyTeachLifterPosB.tyBtn2.bValue				:= FALSE;

			tyP1026McSetTeach.tyMotionStdLifter.tyBtnStop.bRtLk				:= TRUE;
			tyP1026McSetTeach.tyMotionStdLifter.tyBtnJogDown.bRtLk			:= FALSE;
			tyP1026McSetTeach.tyMotionStdLifter.tyBtnJogUp.bRtLk			:= FALSE;
			tyP1026McSetTeach.tyMotionStdLifter.tyBtnOrigin.bRtLk			:= FALSE;
			tyP1026McSetTeach.tyMotionStdLifter.tyBtnMovAbs.bRtLk			:= FALSE;
			tyP1026McSetTeach.tyMotionStdLifter.tyBtnMovRel.bRtLk			:= FALSE;

			tyP1026McSetTeach.tyTeachLifterPosA.tyBtn2.bRtLk				:= FALSE;
			tyP1026McSetTeach.tyTeachLifterPosB.tyBtn2.bRtLk				:= FALSE;

		END_IF

	ELSIF (tyP1026McSetTeach.tyMotionStdLifter.tyBtnJogDown.bRtCompl = TRUE) OR (tyP1026McSetTeach.tyMotionStdLifter.tyBtnJogUp.bRtCompl = TRUE) OR (bJogStopLifter = TRUE) THEN
		bJogSlow					:= FALSE;
		bJogFast					:= FALSE;
		fbJogSlowToFastDlyTm.IN		:= FALSE;

		eLifterBtmAct	:= LifterActJogStop;

		IF p_eLifterBtmStat = LifterActJogStop AND p_eLifterBtmStatus = Done THEN
			eLifterBtmAct		:= LifterActIdle;

			bJogStopLifter	:= FALSE;

			tyP1026McSetTeach.tyMotionStdLifter.tyBtnStop.bRtCompl			:= FALSE;
			tyP1026McSetTeach.tyMotionStdLifter.tyBtnJogDown.bRtCompl		:= FALSE;
			tyP1026McSetTeach.tyMotionStdLifter.tyBtnJogUp.bRtCompl			:= FALSE;
			tyP1026McSetTeach.tyMotionStdLifter.tyBtnOrigin.bRtCompl		:= FALSE;
			tyP1026McSetTeach.tyMotionStdLifter.tyBtnMovAbs.bRtCompl		:= FALSE;
			tyP1026McSetTeach.tyMotionStdLifter.tyBtnMovRel.bRtCompl		:= FALSE;

			tyP1026McSetTeach.tyTeachLifterPosA.tyBtn2.bRtCompl				:= FALSE;
			tyP1026McSetTeach.tyTeachLifterPosB.tyBtn2.bRtCompl				:= FALSE;

			tyP1026McSetTeach.tyMotionStdLifter.tyBtnStop.bValue			:= TRUE;
			tyP1026McSetTeach.tyMotionStdLifter.tyBtnJogDown.bValue			:= FALSE;
			tyP1026McSetTeach.tyMotionStdLifter.tyBtnJogUp.bValue			:= FALSE;
			tyP1026McSetTeach.tyMotionStdLifter.tyBtnOrigin.bValue			:= FALSE;
			tyP1026McSetTeach.tyMotionStdLifter.tyBtnMovAbs.bValue			:= FALSE;
			tyP1026McSetTeach.tyMotionStdLifter.tyBtnMovRel.bValue			:= FALSE;

			tyP1026McSetTeach.tyTeachLifterPosA.tyBtn2.bValue				:= FALSE;
			tyP1026McSetTeach.tyTeachLifterPosB.tyBtn2.bValue				:= FALSE;

			tyP1026McSetTeach.tyMotionStdLifter.tyBtnStop.bRtLk				:= TRUE;
			tyP1026McSetTeach.tyMotionStdLifter.tyBtnJogDown.bRtLk			:= FALSE;
			tyP1026McSetTeach.tyMotionStdLifter.tyBtnJogUp.bRtLk			:= FALSE;
			tyP1026McSetTeach.tyMotionStdLifter.tyBtnOrigin.bRtLk			:= FALSE;
			tyP1026McSetTeach.tyMotionStdLifter.tyBtnMovAbs.bRtLk			:= FALSE;
			tyP1026McSetTeach.tyMotionStdLifter.tyBtnMovRel.bRtLk			:= FALSE;

			tyP1026McSetTeach.tyTeachLifterPosA.tyBtn2.bRtLk				:= FALSE;
			tyP1026McSetTeach.tyTeachLifterPosB.tyBtn2.bRtLk				:= FALSE;

		END_IF

	ELSIF tyP1026McSetTeach.tyMotionStdLifter.tyBtnPwr.bRtCompl = TRUE THEN
		tyP1026McSetTeach.tyMotionStdLifter.tyBtnPwr.bRtLk	:= TRUE;

		IF tyP1026McSetTeach.tyMotionStdLifter.tyBtnPwr.bValue = TRUE THEN
			eLifterBtmAct	:= LifterActPwrOn;

			IF p_eLifterBtmStat = LifterActPwrOn AND p_eLifterBtmStatus = Done THEN
				eLifterBtmAct	:= LifterActIdle;

				tyP1026McSetTeach.tyMotionStdLifter.tyBtnPwr.bRtCompl	:= FALSE;
				tyP1026McSetTeach.tyMotionStdLifter.tyBtnPwr.bRtLk		:= FALSE;
			END_IF
		ELSE
			eLifterBtmAct	:= LifterActPwrOff;

			IF p_eLifterBtmStat = LifterActPwrOff AND p_eLifterBtmStatus = Done THEN
				eLifterBtmAct	:= LifterActIdle;

				tyP1026McSetTeach.tyMotionStdLifter.tyBtnPwr.bRtCompl	:= FALSE;
				tyP1026McSetTeach.tyMotionStdLifter.tyBtnPwr.bRtLk		:= FALSE;
			END_IF
		END_IF

	ELSIF tyP1026McSetTeach.tyMotionStdLifter.tyBtnOrigin.bRtCompl = TRUE THEN
		tyP1026McSetTeach.tyMotionStdLifter.tyBtnOrigin.bValue	:= TRUE;
		tyP1026McSetTeach.tyMotionStdLifter.tyBtnStop.bValue	:= FALSE;

		tyP1026McSetTeach.tyMotionStdLifter.tyBtnOrigin.bRtLk	:= TRUE;
		tyP1026McSetTeach.tyMotionStdLifter.tyBtnStop.bRtLk		:= FALSE;

		eLifterBtmAct	:= LifterActHoming;

		IF p_eLifterBtmStat = LifterActHoming AND p_eLifterBtmStatus = Done THEN
			eLifterBtmAct	:= LifterActIdle;

			tyP1026McSetTeach.tyMotionStdLifter.tyBtnOrigin.bRtCompl	:= FALSE;
			tyP1026McSetTeach.tyMotionStdLifter.tyBtnOrigin.bValue		:= FALSE;
			tyP1026McSetTeach.tyMotionStdLifter.tyBtnStop.bValue		:= TRUE;

			tyP1026McSetTeach.tyMotionStdLifter.tyBtnOrigin.bRtLk		:= FALSE;
			tyP1026McSetTeach.tyMotionStdLifter.tyBtnStop.bRtLk			:= TRUE;

		END_IF

	ELSIF tyP1026McSetTeach.tyMotionStdLifter.tyBtnRst.bRtCompl = TRUE THEN
		tyP1026McSetTeach.tyMotionStdLifter.tyBtnRst.bValue	:= TRUE;
		tyP1026McSetTeach.tyMotionStdLifter.tyBtnRst.bRtLk	:= TRUE;

		eLifterBtmAct	:= LifterActRstAxisErr;

		IF p_eLifterBtmStat = LifterActRstAxisErr AND p_eLifterBtmStatus = Done THEN
			eLifterBtmAct	:= LifterActIdle;

			tyP1026McSetTeach.tyMotionStdLifter.tyBtnRst.bRtCompl	:= FALSE;
			tyP1026McSetTeach.tyMotionStdLifter.tyBtnRst.bValue		:= FALSE;
			tyP1026McSetTeach.tyMotionStdLifter.tyBtnRst.bRtLk		:= FALSE;

			fbLmtRstTm.IN	:= FALSE;
		END_IF

	ELSIF tyP1026McSetTeach.tyTeachLifterPosA.tyBtn2.bRtCompl = TRUE THEN
		tyP1026McSetTeach.tyTeachLifterPosA.tyBtn2.bValue		:= TRUE;
		tyP1026McSetTeach.tyMotionStdLifter.tyBtnStop.bValue	:= FALSE;

		tyP1026McSetTeach.tyTeachLifterPosA.tyBtn2.bRtLk		:= TRUE;
		tyP1026McSetTeach.tyMotionStdLifter.tyBtnStop.bRtLk		:= FALSE;

		diMnlLifterNomSpd	:= tyP1026McSetTeach.tyMotionStdLifter.tyNumNomSpd.diValue;

		eLifterBtmAct	:= LifterActGoAPos;

		IF p_eLifterBtmStat = LifterActGoAPos AND p_eLifterBtmStatus = Done THEN
			eLifterBtmAct	:= LifterActIdle;

			tyP1026McSetTeach.tyTeachLifterPosA.tyBtn2.bRtCompl		:= FALSE;
			tyP1026McSetTeach.tyTeachLifterPosA.tyBtn2.bValue		:= FALSE;
			tyP1026McSetTeach.tyMotionStdLifter.tyBtnStop.bValue	:= TRUE;

			tyP1026McSetTeach.tyTeachLifterPosA.tyBtn2.bRtLk		:= FALSE;
			tyP1026McSetTeach.tyMotionStdLifter.tyBtnStop.bRtLk		:= TRUE;
		END_IF

	ELSIF tyP1026McSetTeach.tyTeachLifterPosB.tyBtn2.bRtCompl = TRUE THEN
		tyP1026McSetTeach.tyTeachLifterPosB.tyBtn2.bValue		:= TRUE;
		tyP1026McSetTeach.tyMotionStdLifter.tyBtnStop.bValue	:= FALSE;

		tyP1026McSetTeach.tyTeachLifterPosB.tyBtn2.bRtLk		:= TRUE;
		tyP1026McSetTeach.tyMotionStdLifter.tyBtnStop.bRtLk		:= FALSE;

		diMnlLifterNomSpd	:= tyP1026McSetTeach.tyMotionStdLifter.tyNumNomSpd.diValue;

		eLifterBtmAct		:= LifterActGoBPos;

		IF p_eLifterBtmStat = LifterActGoBPos AND p_eLifterBtmStatus = Done THEN
			eLifterBtmAct	:= LifterActIdle;

			tyP1026McSetTeach.tyTeachLifterPosB.tyBtn2.bRtCompl		:= FALSE;
			tyP1026McSetTeach.tyTeachLifterPosB.tyBtn2.bValue		:= FALSE;
			tyP1026McSetTeach.tyMotionStdLifter.tyBtnStop.bValue	:= TRUE;

			tyP1026McSetTeach.tyTeachLifterPosB.tyBtn2.bRtLk		:= FALSE;
			tyP1026McSetTeach.tyMotionStdLifter.tyBtnStop.bRtLk		:= TRUE;
		END_IF

	ELSIF tyP1026McSetTeach.tyMotionStdLifter.tyBtnMovAbs.bRtCompl = TRUE THEN

		tyP1026McSetTeach.tyMotionStdLifter.tyBtnMovAbs.bValue	:= TRUE;
		tyP1026McSetTeach.tyMotionStdLifter.tyBtnStop.bValue	:= FALSE;

		tyP1026McSetTeach.tyMotionStdLifter.tyBtnMovAbs.bRtLk	:= TRUE;
		tyP1026McSetTeach.tyMotionStdLifter.tyBtnStop.bRtLk		:= FALSE;

		diMnlLifterTargetPos	:= tyP1026McSetTeach.tyMotionStdLifter.tyNumTargetPos.diValue;
		diMnlLifterNomSpd		:= tyP1026McSetTeach.tyMotionStdLifter.tyNumNomSpd.diValue;

		eLifterBtmAct			:= LifterActMovAbs;

		IF p_eLifterBtmStat = LifterActMovAbs AND p_eLifterBtmStatus = Done THEN
			eLifterBtmAct	:= LifterActIdle;

			tyP1026McSetTeach.tyMotionStdLifter.tyBtnMovAbs.bRtCompl	:= FALSE;
			tyP1026McSetTeach.tyMotionStdLifter.tyBtnMovAbs.bValue		:= FALSE;
			tyP1026McSetTeach.tyMotionStdLifter.tyBtnStop.bValue		:= TRUE;

			tyP1026McSetTeach.tyMotionStdLifter.tyBtnMovAbs.bRtLk		:= FALSE;
			tyP1026McSetTeach.tyMotionStdLifter.tyBtnStop.bRtLk			:= TRUE;
		END_IF

	ELSIF tyP1026McSetTeach.tyMotionStdLifter.tyBtnMovRel.bRtCompl = TRUE THEN
		tyP1026McSetTeach.tyMotionStdLifter.tyBtnMovRel.bValue			:= TRUE;
		tyP1026McSetTeach.tyMotionStdLifter.tyBtnStop.bValue			:= FALSE;

		tyP1026McSetTeach.tyMotionStdLifter.tyBtnMovRel.bRtLk			:= TRUE;
		tyP1026McSetTeach.tyMotionStdLifter.tyBtnStop.bRtLk				:= FALSE;

		diMnlLifterStepSize		:= tyP1026McSetTeach.tyMotionStdLifter.tyNumStepSize.diValue;
		diMnlLifterNomSpd		:= tyP1026McSetTeach.tyMotionStdLifter.tyNumNomSpd.diValue;

		eLifterBtmAct		:= LifterActMovRel;

		IF p_eLifterBtmStat = LifterActMovRel AND p_eLifterBtmStatus = Done THEN
			eLifterBtmAct	:= LifterActIdle;

			tyP1026McSetTeach.tyMotionStdLifter.tyBtnMovRel.bRtCompl		:= FALSE;
			tyP1026McSetTeach.tyMotionStdLifter.tyBtnMovRel.bValue			:= FALSE;
			tyP1026McSetTeach.tyMotionStdLifter.tyBtnStop.bValue			:= TRUE;

			tyP1026McSetTeach.tyMotionStdLifter.tyBtnMovRel.bRtLk			:= FALSE;
			tyP1026McSetTeach.tyMotionStdLifter.tyBtnStop.bRtLk				:= TRUE;

		END_IF

	ELSIF (tyP1026McSetTeach.tyMotionStdLifter.tyBtnJogDown.bValue = TRUE) AND (fbJogSlowToFastDlyTm.Q = FALSE) AND (bJogSlow = FALSE) THEN
		tyP1026McSetTeach.tyMotionStdLifter.tyBtnStop.bValue				:= FALSE;
		tyP1026McSetTeach.tyMotionStdLifter.tyBtnStop.bRtLk				:= FALSE;

		fbJogSlowToFastDlyTm.IN		:= TRUE;

		diMnlLifterJogSpd	:= tyP1026McSetTeach.tyMotionStdLifter.tyNumSlwSpd.diValue;

		eLifterBtmAct		:= LifterActJogDown;

		IF p_eLifterBtmStat = LifterActJogDown AND p_eLifterBtmStatus = Done THEN

			eLifterBtmAct	:= LifterActIdle;
			bJogSlow				:= TRUE;

		ELSIF p_eLifterBtmStatus = Error THEN

			fbJogSlowToFastDlyTm.IN	:= FALSE;
			bJogSlow				:= TRUE;

		END_IF

	ELSIF (tyP1026McSetTeach.tyMotionStdLifter.tyBtnJogDown.bValue = TRUE) AND (fbJogSlowToFastDlyTm.Q = TRUE) AND (bJogFast = FALSE) THEN
		tyP1026McSetTeach.tyMotionStdLifter.tyBtnStop.bValue					:= FALSE;
		tyP1026McSetTeach.tyMotionStdLifter.tyBtnStop.bRtLk					:= FALSE;

		fbJogSlowToFastDlyTm.IN		:= TRUE;

		diMnlLifterJogSpd	:= tyP1026McSetTeach.tyMotionStdLifter.tyNumNomSpd.diValue;

		eLifterBtmAct		:= LifterActJogDown;

		IF p_eLifterBtmStat = LifterActJogDown AND p_eLifterBtmStatus = Done THEN
			eLifterBtmAct	:= LifterActIdle;
			bJogFast				:= TRUE;
		ELSIF p_eLifterBtmStatus = Error THEN
			fbJogSlowToFastDlyTm.IN	:= FALSE;
			bJogFast				:= TRUE;
		END_IF

	ELSIF (tyP1026McSetTeach.tyMotionStdLifter.tyBtnJogUp.bValue = TRUE) AND (fbJogSlowToFastDlyTm.Q = FALSE) AND (bJogSlow = FALSE) THEN
		tyP1026McSetTeach.tyMotionStdLifter.tyBtnStop.bValue				:= FALSE;
		tyP1026McSetTeach.tyMotionStdLifter.tyBtnStop.bRtLk				:= FALSE;

		fbJogSlowToFastDlyTm.IN		:= TRUE;

		diMnlLifterJogSpd	:= tyP1026McSetTeach.tyMotionStdLifter.tyNumSlwSpd.diValue;

		eLifterBtmAct		:= LifterActJogUp;

		IF p_eLifterBtmStat = LifterActJogUp AND p_eLifterBtmStatus = Done THEN
			eLifterBtmAct	:= LifterActIdle;
			bJogSlow				:= TRUE;

		ELSIF p_eLifterBtmStatus = Error THEN
			fbJogSlowToFastDlyTm.IN	:= FALSE;
			bJogSlow				:= TRUE;
		END_IF

	ELSIF (tyP1026McSetTeach.tyMotionStdLifter.tyBtnJogUp.bValue = TRUE) AND (fbJogSlowToFastDlyTm.Q = TRUE) AND (bJogFast = FALSE) THEN

		tyP1026McSetTeach.tyMotionStdLifter.tyBtnStop.bValue				:= FALSE;
		tyP1026McSetTeach.tyMotionStdLifter.tyBtnStop.bRtLk					:= FALSE;

		fbJogSlowToFastDlyTm.IN		:= TRUE;

		diMnlLifterJogSpd	:= tyP1026McSetTeach.tyMotionStdLifter.tyNumNomSpd.diValue;

		eLifterBtmAct		:= LifterActJogUp;

		IF p_eLifterBtmStat = LifterActJogUp AND p_eLifterBtmStatus = Done THEN
			eLifterBtmAct	:= LifterActIdle;
			bJogFast	:= TRUE;

		ELSIF p_eLifterBtmStatus = Error THEN
			fbJogSlowToFastDlyTm.IN	:= FALSE;
			bJogFast				:= TRUE;
		END_IF
	END_IF

	IF tyP1026McSetTeach.tyInOutletShutterFB.tyBtnOpen.bRtCompl = TRUE THEN
		tyP1026McSetTeach.tyInOutletShutterFB.tyBtnOpen.bRtCompl	:= FALSE;

		tyP1026McSetTeach.tyInOutletShutterFB.tyBtnOpen.bValue	:= TRUE;
		tyP1026McSetTeach.tyInOutletShutterFB.tyBtnClose.bValue	:= FALSE;

	ELSIF tyP1026McSetTeach.tyInOutletShutterFB.tyBtnClose.bRtCompl = TRUE THEN
		tyP1026McSetTeach.tyInOutletShutterFB.tyBtnClose.bRtCompl	:= FALSE;

		tyP1026McSetTeach.tyInOutletShutterFB.tyBtnClose.bValue	:= TRUE;
		tyP1026McSetTeach.tyInOutletShutterFB.tyBtnOpen.bValue	:= FALSE;
	END_IF

	IF tyP1026McSetTeach.tyInOutletShutterFB.tyBtnOpen.bValue = TRUE THEN
		eInShutterAct	:= PneuActRet;
		eOutShutterAct	:= PneuActRet;

		IF (p_eInShutterStat = PneuActRet AND p_eInShutterStatus = Done)
			AND (p_eOutShutterStat = PneuActRet AND p_eOutShutterStatus = Done)
			THEN
			eInShutterAct	:= PneuActIdle;
			eOutShutterAct	:= PneuActIdle;
			tyP1026McSetTeach.tyInOutletShutterFB.tyBtnOpen.bValue	:= FALSE;
		ELSIF p_eInShutterStatus = Error OR p_eOutShutterStatus = Error THEN
			tyP1026McSetTeach.tyInOutletShutterFB.tyBtnOpen.bValue	:= FALSE;
		END_IF

	ELSIF tyP1026McSetTeach.tyInOutletShutterFB.tyBtnClose.bValue = TRUE THEN
		eInShutterAct	:= PneuActExt;
		eOutShutterAct	:= PneuActExt;
		IF (p_eInShutterStat = PneuActExt AND p_eInShutterStatus = Done)
			AND (p_eOutShutterStat = PneuActExt AND p_eOutShutterStatus = Done)
			THEN
			eInShutterAct	:= PneuActIdle;
			eOutShutterAct	:= PneuActIdle;
			tyP1026McSetTeach.tyInOutletShutterFB.tyBtnClose.bValue := FALSE;
		ELSIF p_eInShutterStatus = Error OR p_eOutShutterStatus = Error THEN
			tyP1026McSetTeach.tyInOutletShutterFB.tyBtnClose.bValue := FALSE;
		END_IF
	END_IF

	//bypass curtain sensor
	IF bTeachLifterPosA OR bTeachLifterPosB THEN
		bBypCurtainSen			:= tyP1026McSetTeach.tyTeachLifterPosA.tyBtn4.bValue OR tyP1026McSetTeach.tyTeachLifterPosB.tyBtn4.bValue;
		bBypCurtainPBLED		:= tyP1026McSetTeach.tyTeachLifterPosA.tyBtn4.bValue OR tyP1026McSetTeach.tyTeachLifterPosB.tyBtn4.bValue;
	END_IF

END_ACTION
```

#### Act_OptP1026LifterUpdtDat.st
```iecst
ACTION Act_OptP1026LifterUpdtDat:

	tyP1026McSetTeach.tyMotionStdLifter.tyNumCurrPos.diValue		:= p_diLifterBtmActualPos;
	tyP1026McSetTeach.tyMotionStdLifter.tyNumErrCode.diValue		:= UDINT_TO_DINT(p_udiLifterBtmAxisErrID);
	tyP1026McSetTeach.tyMotionStdLifter.tyBitmapPwr.usiValueIdx		:= BOOL_TO_USINT(p_bLifterBtmPwrOn);
	tyP1026McSetTeach.tyMotionStdLifter.tyBitmapRst.usiValueIdx		:= BOOL_TO_USINT(NOT p_bLifterBtmAxisErr);
	tyP1026McSetTeach.tyMotionStdLifter.tyBitmapOrigin.usiValueIdx	:= BOOL_TO_USINT(p_bLifterBtmIsHomed);
	tyP1026McSetTeach.tyMotionStdLifter.tyBtnUpLmtSen.bValue		:= p_bLifterBtmUpSen;
	tyP1026McSetTeach.tyMotionStdLifter.tyBtnDownLmtSen.bValue		:= p_bLifterBtmDownSen;

	//Machine Bitmap
	IF   (p_tyNtParamCurr.eProjMag = LDMagDual AND p_tyNtParamCurr.bMagAutoVerifyPrep = FALSE)
		OR (p_tyNtParamCurr.eProjMag = LDMagTriple AND p_tyNtParamCurr.bMagAutoVerifyPrep = FALSE)
		OR (p_tyNtParamCurr.eProjMag = LDMagDual AND p_tyNtParamCurr.bMagAutoVerifyPrep = TRUE)
		THEN
		IF p_bLifterBtmIsHomed = TRUE THEN

			IF p_diLifterBtmActualPos <= (p_tyNtParamCurr.tyUILifterTargetPos.diMax / 3) THEN
				tyP1026McSetTeach.tyMotionStdLifter.tyBitmapMc.uiValueIdx 	:= 2;
			ELSIF p_diLifterBtmActualPos <= (p_tyNtParamCurr.tyUILifterTargetPos.diMax / 3 * 2) THEN
				tyP1026McSetTeach.tyMotionStdLifter.tyBitmapMc.uiValueIdx 	:= 3;
			ELSE
				tyP1026McSetTeach.tyMotionStdLifter.tyBitmapMc.uiValueIdx 	:= 4;
			END_IF

		ELSE
			tyP1026McSetTeach.tyMotionStdLifter.tyBitmapMc.uiValueIdx	:= 2;
		END_IF

	ELSIF p_tyNtParamCurr.eProjMag = LDMagTriple AND p_tyNtParamCurr.bMagAutoVerifyPrep = TRUE
		THEN
		IF p_bLifterBtmIsHomed = TRUE THEN

			IF p_diLifterBtmActualPos <= (p_tyNtParamCurr.tyUILifterTargetPos.diMax / 3) THEN
				tyP1026McSetTeach.tyMotionStdLifter.tyBitmapMc.uiValueIdx 	:= 23;
			ELSIF p_diLifterBtmActualPos <= (p_tyNtParamCurr.tyUILifterTargetPos.diMax / 3 * 2) THEN
				tyP1026McSetTeach.tyMotionStdLifter.tyBitmapMc.uiValueIdx 	:= 24;
			ELSE
				tyP1026McSetTeach.tyMotionStdLifter.tyBitmapMc.uiValueIdx 	:= 25;
			END_IF

		ELSE
			tyP1026McSetTeach.tyMotionStdLifter.tyBitmapMc.uiValueIdx	:= 23;
		END_IF

	ELSIF p_tyNtParamCurr.eProjMag = LDMagQuadruple AND p_tyNtParamCurr.bMagAutoVerifyPrep = TRUE
		THEN
		IF p_bLifterBtmIsHomed = TRUE THEN

			IF p_diLifterBtmActualPos <= (p_tyNtParamCurr.tyUILifterTargetPos.diMax / 3) THEN
				tyP1026McSetTeach.tyMotionStdLifter.tyBitmapMc.uiValueIdx 	:= 27;
			ELSIF p_diLifterBtmActualPos <= (p_tyNtParamCurr.tyUILifterTargetPos.diMax / 3 * 2) THEN
				tyP1026McSetTeach.tyMotionStdLifter.tyBitmapMc.uiValueIdx 	:= 28;
			ELSE
				tyP1026McSetTeach.tyMotionStdLifter.tyBitmapMc.uiValueIdx 	:= 29;
			END_IF

		ELSE
			tyP1026McSetTeach.tyMotionStdLifter.tyBitmapMc.uiValueIdx	:= 27;
		END_IF
	END_IF

	IF p_tyNtParamCurr.eProjMag = LDMagTriple AND p_tyNtParamCurr.bProjLifterMagPlatform THEN
		IF 	tyP1026McSetTeach.tyMotionStdLifter.tyBitmapMc.uiValueIdx < 400 THEN
			tyP1026McSetTeach.tyMotionStdLifter.tyBitmapMc.uiValueIdx	:= tyP1031MagSetTeach.tyMotionStdLifter.tyBitmapMc.uiValueIdx + 400;
		END_IF
	ELSIF (p_tyNtParamCurr.eProjMag = LDMagDual OR p_tyNtParamCurr.eProjMag = LDMagTriple) AND p_tyNtParamCurr.bProjMotorizedPullerPrep = FALSE THEN
		IF 	tyP1026McSetTeach.tyMotionStdLifter.tyBitmapMc.uiValueIdx < 200 THEN
			tyP1026McSetTeach.tyMotionStdLifter.tyBitmapMc.uiValueIdx	:= tyP1026McSetTeach.tyMotionStdLifter.tyBitmapMc.uiValueIdx + 200;
		END_IF
	ELSIF p_tyNtParamCurr.eProjMag = LDMagDual AND p_tyNtParamCurr.bProjMotorizedPullerPrep THEN
		IF p_tyNtParamCurr.sJobNo = '2023-0258A01' THEN
			tyP1026McSetTeach.tyMotionStdLifter.tyBitmapMc.uiValueIdx	:= tyP1026McSetTeach.tyMotionStdLifter.tyBitmapMc.uiValueIdx + 444-2;
		END_IF

	ELSIF p_tyNtParamCurr.eProjMag = LDMagTriple AND p_tyNtParamCurr.bMagAutoVerifyPrep = FALSE AND p_tyNtParamCurr.bProjMotorizedPullerPrep = TRUE
		THEN
		IF 	tyP1026McSetTeach.tyMotionStdLifter.tyBitmapMc.uiValueIdx < 300 THEN
			tyP1026McSetTeach.tyMotionStdLifter.tyBitmapMc.uiValueIdx	:= tyP1026McSetTeach.tyMotionStdLifter.tyBitmapMc.uiValueIdx + 300;
		END_IF
	END_IF

END_ACTION
```

#### Act_OptP1026LifterRstMnl.st
```iecst
ACTION Act_OptP1026LifterRstMnl:

	IF EDGEPOS((bManualMod = FALSE) OR (p_eLifterBtmStatus = Error)) THEN

		bJogSlow				:= FALSE;
		bJogFast				:= FALSE;
		fbJogSlowToFastDlyTm.IN	:= FALSE;

		tyP1026McSetTeach.tyMotionStdLifter.tyBtnPwr.bRtCompl			:= FALSE;
		tyP1026McSetTeach.tyMotionStdLifter.tyBtnStop.bRtCompl			:= FALSE;
		tyP1026McSetTeach.tyMotionStdLifter.tyBtnOrigin.bRtCompl		:= FALSE;
		tyP1026McSetTeach.tyMotionStdLifter.tyBtnRst.bRtCompl			:= FALSE;
		tyP1026McSetTeach.tyMotionStdLifter.tyBtnMovAbs.bRtCompl		:= FALSE;
		tyP1026McSetTeach.tyMotionStdLifter.tyBtnMovRel.bRtCompl		:= FALSE;
		tyP1026McSetTeach.tyMotionStdLifter.tyBtnJogUp.bRtCompl			:= FALSE;
		tyP1026McSetTeach.tyMotionStdLifter.tyBtnJogDown.bRtCompl		:= FALSE;

		tyP1026McSetTeach.tyTeachLifterPosA.tyBtn2.bRtCompl				:= FALSE;
		tyP1026McSetTeach.tyTeachLifterPosB.tyBtn2.bRtCompl				:= FALSE;

		tyP1026McSetTeach.tyMotionStdLifter.tyBtnPwr.bValue				:= FALSE;
		tyP1026McSetTeach.tyMotionStdLifter.tyBtnStop.bValue			:= TRUE;
		tyP1026McSetTeach.tyMotionStdLifter.tyBtnOrigin.bValue			:= FALSE;
		tyP1026McSetTeach.tyMotionStdLifter.tyBtnRst.bValue				:= FALSE;
		tyP1026McSetTeach.tyMotionStdLifter.tyBtnMovAbs.bValue			:= FALSE;
		tyP1026McSetTeach.tyMotionStdLifter.tyBtnMovRel.bValue			:= FALSE;
		tyP1026McSetTeach.tyMotionStdLifter.tyBtnJogUp.bValue			:= FALSE;
		tyP1026McSetTeach.tyMotionStdLifter.tyBtnJogDown.bValue			:= FALSE;

		tyP1026McSetTeach.tyTeachLifterPosA.tyBtn2.bValue				:= FALSE;
		tyP1026McSetTeach.tyTeachLifterPosB.tyBtn2.bValue				:= FALSE;

		tyP1026McSetTeach.tyMotionStdLifter.tyBtnPwr.bRtLk				:= FALSE;
		tyP1026McSetTeach.tyMotionStdLifter.tyBtnStop.bRtLk				:= TRUE;
		tyP1026McSetTeach.tyMotionStdLifter.tyBtnOrigin.bRtLk			:= FALSE;
		tyP1026McSetTeach.tyMotionStdLifter.tyBtnRst.bRtLk				:= FALSE;
		tyP1026McSetTeach.tyMotionStdLifter.tyBtnMovAbs.bRtLk			:= FALSE;
		tyP1026McSetTeach.tyMotionStdLifter.tyBtnMovRel.bRtLk			:= FALSE;
		tyP1026McSetTeach.tyMotionStdLifter.tyBtnJogUp.bRtLk			:= FALSE;
		tyP1026McSetTeach.tyMotionStdLifter.tyBtnJogDown.bRtLk			:= FALSE;

		tyP1026McSetTeach.tyTeachLifterPosA.tyBtn2.bRtLk				:= FALSE;
		tyP1026McSetTeach.tyTeachLifterPosB.tyBtn2.bRtLk				:= FALSE;

		tyP1026McSetTeach.tyMotionStdLifter.tyBtnPwr.uiMaskRtStat		:= TRUE;
		tyP1026McSetTeach.tyMotionStdLifter.tyBtnOrigin.uiMaskRtStat	:= FALSE;
		tyP1026McSetTeach.tyMotionStdLifter.tyBtnRst.uiMaskRtStat		:= TRUE;
		tyP1026McSetTeach.tyMotionStdLifter.tyBtnMovAbs.uiMaskRtStat	:= FALSE;
		tyP1026McSetTeach.tyMotionStdLifter.tyBtnMovRel.uiMaskRtStat	:= FALSE;
		tyP1026McSetTeach.tyMotionStdLifter.tyBtnJogUp.uiMaskRtStat		:= FALSE;
		tyP1026McSetTeach.tyMotionStdLifter.tyBtnJogDown.uiMaskRtStat	:= FALSE;

		tyP1026McSetTeach.tyTeachLifterPosA.tyBtn2.uiMaskRtStat			:= FALSE;
		tyP1026McSetTeach.tyTeachLifterPosB.tyBtn2.uiMaskRtStat			:= FALSE;

		eInShutterAct	:= PneuActIdle;
		eOutShutterAct	:= PneuActIdle;

		tyP1026McSetTeach.tyInOutletShutterFB.tyBtnClose.bRtCompl	:= FALSE;
		tyP1026McSetTeach.tyInOutletShutterFB.tyBtnClose.bValue	:= FALSE;
		tyP1026McSetTeach.tyInOutletShutterFB.tyBtnOpen.bRtCompl	:= FALSE;
		tyP1026McSetTeach.tyInOutletShutterFB.tyBtnOpen.bValue	:= FALSE;
	END_IF

END_ACTION
```

#### Act_EntP1027Disp.st
```iecst
ACTION Act_EntP1027Disp:

	//Access Address
	p_tyC0004Navi ACCESS ADR(tyP1027McSetUSBSetting.tyNaviBack);

	p_tyC0005Main ACCESS ADR(tyCommon.tyMain);

	p_tyC0006Set ACCESS ADR(tyCommon.tySet);

	p_tyC0007Notif ACCESS ADR(tyCommon.tyNotif);

	p_tyC0008MsgBox ACCESS ADR(tyP1027McSetUSBSetting.tyMsgBoxHide);

	p_tyC0009Info ACCESS ADR(tyCommon.tyInfo);

	p_tyP1027McSetUSBSetting ACCESS ADR(tyP1027McSetUSBSetting.tyUSBSet);

	//Backup Param
	tyP1027McSetUSBSetting.tyUSBSetBkUp	:= tyP1027McSetUSBSetting.tyUSBSet;

END_ACTION
```

#### Act_ExitP1027.st
```iecst
ACTION Act_ExitP1027:

	IF tyCommon.tySet.tyBtnSave.uiMaskRtStat.0 = FALSE THEN
		usiChgPage	:= 1;

	ELSE

		p_tyC0008MsgBox ACCESS ADR(tyP1027McSetUSBSetting.tyMsgBoxExitAsk);

		IF tyP1027McSetUSBSetting.tyMsgBoxExitAsk.tyBtnYes.bRtCompl = TRUE THEN
			tyP1027McSetUSBSetting.tyMsgBoxExitAsk.tyBtnYes.bRtCompl	:= FALSE;
			tyP1027McSetUSBSetting.tyMsgBoxExitAsk.tyBtnYes.bValue	:= FALSE;

			p_tyC0008MsgBox ACCESS ADR(tyP1027McSetUSBSetting.tyMsgBoxHide);

			//Restore Param
			tyP1027McSetUSBSetting.tyUSBSet	:= tyP1027McSetUSBSetting.tyUSBSetBkUp;

			fUIInRtStatOff(ADR(tyCommon.tySet.tyBtnSave.uiMaskRtStat));

			usiChgPage	:= 1;

		ELSIF tyP1027McSetUSBSetting.tyMsgBoxExitAsk.tyBtnNo.bRtCompl = TRUE THEN
			tyP1027McSetUSBSetting.tyMsgBoxExitAsk.tyBtnNo.bRtCompl	:= FALSE;
			tyP1027McSetUSBSetting.tyMsgBoxExitAsk.tyBtnNo.bValue	:= FALSE;

			p_tyC0008MsgBox ACCESS ADR(tyP1027McSetUSBSetting.tyMsgBoxHide);

			eChgPage	:= eCurrPage;
			usiChgPage	:= 0;

		END_IF

	END_IF

END_ACTION
```

#### Act_OptP1027Keypad.st
```iecst
ACTION Act_OptP1027Keypad:

	IF fUIOutRtStatTPIsOpen(ADR(tyP1027McSetUSBSetting.tyUSBSet.tyVID.uiRtStat)) = TRUE THEN
		tyProperty.tyKeypad.tyStringTitle.sKeypadTitle			:= tyP1027McSetUSBSetting.tyUSBSet.tyVID.sKeypadTitle;

	ELSIF fUIOutRtStatTPIsOpen(ADR(tyP1027McSetUSBSetting.tyUSBSet.tyPID.uiRtStat)) = TRUE THEN
		tyProperty.tyKeypad.tyStringTitle.sKeypadTitle			:= tyP1027McSetUSBSetting.tyUSBSet.tyPID.sKeypadTitle;

	END_IF

END_ACTION
```

#### Act_OptP1027Navi.st
```iecst
ACTION Act_OptP1027Navi:

	IF tyP1027McSetUSBSetting.tyNaviBack.tyBtnBack.bRtCompl = TRUE THEN
		tyP1027McSetUSBSetting.tyNaviBack.tyBtnBack.bRtCompl	:= FALSE;

		eChgPage	:= UIP1020McSetNavi;

	END_IF

END_ACTION
```

#### Act_OptP1027Save.st
```iecst
ACTION Act_OptP1027Save:

	//Reset button
	bResetButton	:= tyP1027McSetUSBSetting.tyUSBSet.tyBtnReset.bValue;		// ADD

	IF p_eUSBRdrStatus = Error THEN
		tyP1027McSetUSBSetting.tyUSBSet.tyBitError.usiValueIdx	:= 2;
	ELSE
		tyP1027McSetUSBSetting.tyUSBSet.tyBitError.usiValueIdx	:= 0;
	END_IF

	IF tyP1027McSetUSBSetting.tyUSBSet.tyVID.bRtCompl OR tyP1027McSetUSBSetting.tyUSBSet.tyPID.bRtCompl THEN

		fUIInRtStatHide(ADR(tyCommon.tySet.tyBtnSave.uiMaskRtStat));

		tyP1027McSetUSBSetting.tyUSBSet.tyVID.bRtCompl := FALSE;
		tyP1027McSetUSBSetting.tyUSBSet.tyPID.bRtCompl := FALSE;

	END_IF

//	eUSBRdrAct	:= USBRdrActIdle;                               //ADD

	IF tyCommon.tySet.tyBtnSave.bRtCompl = TRUE THEN

		fUIInRtStatOff(ADR(tyCommon.tySet.tyBtnSave.uiMaskRtStat));

		tyMcParamWr.diVID	:=  tyP1027McSetUSBSetting.tyUSBSet.tyVID.diValue;
		tyMcParamWr.diPID	:=  tyP1027McSetUSBSetting.tyUSBSet.tyPID.diValue;

		eMcParamAct	:= McParamActWrite;

		IF p_eMcParamStat = McParamActWrite AND p_eMcParamStatus = Done THEN

			eMcParamAct	:= McParamActIdle;
			eUSBRdrAct	:= USBRdrActDetectDev;

			//Update BackUp Param
			tyP1027McSetUSBSetting.tyUSBSetBkUp	:= tyP1027McSetUSBSetting.tyUSBSet;
			tyCommon.tySet.tyBtnSave.bRtCompl	:= FALSE;

		END_IF
	END_IF

	IF (p_eUSBRdrStat = USBRdrActDetectDev OR p_eUSBRdrStat = USBRdrActSafetyRmv) AND p_eUSBRdrStatus = Done THEN
		eUSBRdrAct := USBRdrActIdle;
	END_IF

//		ELSIF p_eMcParamStatus = Error OR p_eUSBRdrStatus = Error THEN
//			p_tyC0008MsgBox ACCESS ADR(tyP1027McSetUSBSetting.tyMsgBoxSaveErr);
//
//			IF tyP1027McSetUSBSetting.tyMsgBoxSaveErr.tyBtnNo.bRtCompl = TRUE THEN
//				tyP1027McSetUSBSetting.tyMsgBoxSaveErr.tyBtnNo.bRtCompl 	:= FALSE;
//				tyP1027McSetUSBSetting.tyMsgBoxSaveErr.tyBtnNo.bValue	:= FALSE;
//
//				p_tyC0008MsgBox ACCESS ADR(tyP1027McSetUSBSetting.tyMsgBoxHide);
//
//				//Restore Param
//				tyP1027McSetUSBSetting.tyUSBSet	:= tyP1027McSetUSBSetting.tyUSBSetBkUp;
//
//				tyMcParamWr								:= p_tyMcParamCurr;
//
//				tyCommon.tySet.tyBtnSave.bRtCompl 	:= FALSE;
//				fUIInRtStatOff(ADR(tyCommon.tySet.tyBtnSave.uiMaskRtStat));
//				eUSBRdrAct	:= USBRdrActIdle;
//				//p_eUSBRdrStatus := Idle;
//			END_IF

	//	END_IF

	//	eUSBRdrAct	:= USBRdrActDetectDev;

	//	IF p_eUSBRdrStat = USBRdrActDetectDev AND p_eUSBRdrStatus = Done THEN
	//		eUSBRdrAct := USBRdrActIdle;

	//	ELSE
	//		eUSBRdrAct := USBRdrActIdle;

	//	END_IF

//	END_IF

END_ACTION
```

#### Act_EntP1028Disp.st
```iecst
ACTION Act_EntP1028Disp:

	//Access Address
	p_tyC0004Navi ACCESS ADR(tyP1028McSetRS232Setting.tyNaviBack);

	p_tyC0005Main ACCESS ADR(tyCommon.tyMain);

	p_tyC0006Set ACCESS ADR(tyCommon.tySet);

	p_tyC0007Notif ACCESS ADR(tyCommon.tyNotif);

	p_tyC0008MsgBox ACCESS ADR (tyP1028McSetRS232Setting.tyMsgBoxHide);

	p_tyC0009Info ACCESS ADR(tyCommon.tyInfo);

	p_tyP1028McSetRS232Setting ACCESS ADR(tyP1028McSetRS232Setting.tyRS232Set);

	//Backup Param
	tyP1028McSetRS232Setting.tyRS232SetBkUp	:= tyP1028McSetRS232Setting.tyRS232Set;

END_ACTION
```

#### Act_ExitP1028.st
```iecst
ACTION Act_ExitP1028:

	IF tyCommon.tySet.tyBtnSave.uiMaskRtStat.0 = FALSE THEN
		usiChgPage	:= 1;

	ELSE

		p_tyC0008MsgBox ACCESS ADR(tyP1028McSetRS232Setting.tyMsgBoxExitAsk);

		IF tyP1028McSetRS232Setting.tyMsgBoxExitAsk.tyBtnYes.bRtCompl = TRUE THEN
			tyP1028McSetRS232Setting.tyMsgBoxExitAsk.tyBtnYes.bRtCompl	:= FALSE;
			tyP1028McSetRS232Setting.tyMsgBoxExitAsk.tyBtnYes.bValue	:= FALSE;

			p_tyC0008MsgBox ACCESS ADR(tyP1028McSetRS232Setting.tyMsgBoxHide);

			//Restore Param
			tyP1028McSetRS232Setting.tyRS232Set	:= tyP1028McSetRS232Setting.tyRS232SetBkUp;

			fUIInRtStatOff(ADR(tyCommon.tySet.tyBtnSave.uiMaskRtStat));

			usiChgPage	:= 1;

		ELSIF tyP1028McSetRS232Setting.tyMsgBoxExitAsk.tyBtnNo.bRtCompl = TRUE THEN
			tyP1028McSetRS232Setting.tyMsgBoxExitAsk.tyBtnNo.bRtCompl	:= FALSE;
			tyP1028McSetRS232Setting.tyMsgBoxExitAsk.tyBtnNo.bValue		:= FALSE;

			p_tyC0008MsgBox ACCESS ADR(tyP1028McSetRS232Setting.tyMsgBoxHide);

			eChgPage	:= eCurrPage;
			usiChgPage	:= 0;

		END_IF

	END_IF

END_ACTION
```

#### Act_OptP1028Navi.st
```iecst
ACTION Act_OptP1028Navi:

	tyP1028McSetRS232Setting.tyNaviBack.tyBtnBack.bRtLk	:= tyCommon.tySet.tyBtnSave.bRtCompl;

	IF tyP1028McSetRS232Setting.tyNaviBack.tyBtnBack.bRtCompl = TRUE THEN
		tyP1028McSetRS232Setting.tyNaviBack.tyBtnBack.bRtCompl	:= FALSE;

		eChgPage	:= UIP1020McSetNavi;

	END_IF

END_ACTION
```

#### Act_OptP1028Save.st
```iecst
ACTION Act_OptP1028Save:

	IF tyP1028McSetRS232Setting.tyRS232Set.tyNumStartCode1.bRtCompl OR tyP1028McSetRS232Setting.tyRS232Set.tyNumStartCode2.bRtCompl
		OR tyP1028McSetRS232Setting.tyRS232Set.tyNumEndCode1.bRtCompl OR  tyP1028McSetRS232Setting.tyRS232Set.tyNumEndCode2.bRtCompl THEN

		fUIInRtStatHide(ADR(tyCommon.tySet.tyBtnSave.uiMaskRtStat));

		tyP1028McSetRS232Setting.tyRS232Set.tyNumStartCode1.bRtCompl := FALSE;
		tyP1028McSetRS232Setting.tyRS232Set.tyNumStartCode2.bRtCompl := FALSE;
		tyP1028McSetRS232Setting.tyRS232Set.tyNumEndCode1.bRtCompl	 := FALSE;
		tyP1028McSetRS232Setting.tyRS232Set.tyNumEndCode2.bRtCompl	 := FALSE;

	END_IF

	IF tyCommon.tySet.tyBtnSave.bRtCompl = TRUE THEN

		tyMcParamWr.diRS232StartCode1	:=  tyP1028McSetRS232Setting.tyRS232Set.tyNumStartCode1.diValue;
		tyMcParamWr.diRS232StartCode2	:=  tyP1028McSetRS232Setting.tyRS232Set.tyNumStartCode2.diValue;
		tyMcParamWr.diRS232EndCode1	    :=  tyP1028McSetRS232Setting.tyRS232Set.tyNumEndCode1.diValue;
		tyMcParamWr.diRS232EndCode2		:=  tyP1028McSetRS232Setting.tyRS232Set.tyNumEndCode2.diValue;

		eMcParamAct	:= McParamActWrite;

		IF p_eMcParamStat = McParamActWrite AND p_eMcParamStatus = Done THEN
			eMcParamAct	:= McParamActIdle;

			//Update BackUp Param
			tyP1028McSetRS232Setting.tyRS232SetBkUp	:= tyP1028McSetRS232Setting.tyRS232Set;

			tyCommon.tySet.tyBtnSave.bRtCompl	:= FALSE;
			fUIInRtStatOff(ADR(tyCommon.tySet.tyBtnSave.uiMaskRtStat));

		ELSIF p_eMcParamStatus = Error THEN
			p_tyC0008MsgBox ACCESS ADR(tyP1028McSetRS232Setting.tyMsgBoxSaveErr);

			IF tyP1028McSetRS232Setting.tyMsgBoxSaveErr.tyBtnNo.bRtCompl = TRUE THEN
				tyP1028McSetRS232Setting.tyMsgBoxSaveErr.tyBtnNo.bRtCompl 	:= FALSE;
				tyP1028McSetRS232Setting.tyMsgBoxSaveErr.tyBtnNo.bValue	:= FALSE;

				p_tyC0008MsgBox ACCESS ADR(tyP1028McSetRS232Setting.tyMsgBoxHide);

				//Restore Param
				tyP1028McSetRS232Setting.tyRS232Set	:= tyP1028McSetRS232Setting.tyRS232SetBkUp;

				tyMcParamWr		:= p_tyMcParamCurr;

				tyCommon.tySet.tyBtnSave.bRtCompl 	:= FALSE;
				fUIInRtStatOff(ADR(tyCommon.tySet.tyBtnSave.uiMaskRtStat));

			END_IF

		END_IF

	END_IF

END_ACTION
```

#### Act_OptP1028Keypad.st
```iecst
ACTION Act_OptP1028Keypad:

	IF fUIOutRtStatTPIsOpen(ADR(tyP1028McSetRS232Setting.tyRS232Set.tyNumStartCode1.uiRtStat)) = TRUE THEN
		tyProperty.tyKeypad.tyStringTitle.sKeypadTitle	:= tyP1028McSetRS232Setting.tyRS232Set.tyNumStartCode1.sKeypadTitle;

	ELSIF fUIOutRtStatTPIsOpen(ADR(tyP1028McSetRS232Setting.tyRS232Set.tyNumStartCode2.uiRtStat)) = TRUE THEN
		tyProperty.tyKeypad.tyStringTitle.sKeypadTitle	:= tyP1028McSetRS232Setting.tyRS232Set.tyNumStartCode2.sKeypadTitle;

	ELSIF fUIOutRtStatTPIsOpen(ADR(tyP1028McSetRS232Setting.tyRS232Set.tyNumEndCode1.uiRtStat)) = TRUE THEN
		tyProperty.tyKeypad.tyStringTitle.sKeypadTitle	:= tyP1028McSetRS232Setting.tyRS232Set.tyNumEndCode1.sKeypadTitle;

	ELSIF fUIOutRtStatTPIsOpen(ADR(tyP1028McSetRS232Setting.tyRS232Set.tyNumEndCode2.uiRtStat)) = TRUE THEN
		tyProperty.tyKeypad.tyStringTitle.sKeypadTitle	:= tyP1028McSetRS232Setting.tyRS232Set.tyNumEndCode2.sKeypadTitle;

	END_IF

END_ACTION
```

#### Act_EntP1030Disp.st
```iecst
ACTION Act_EntP1030Disp:

	//Access Address
	p_tyC0005Main ACCESS ADR(tyCommon.tyMain);

	p_tyC0007Notif ACCESS ADR(tyCommon.tyNotif);

	p_tyC0008MsgBox ACCESS ADR(tyP1030MagSet.tyMsgBoxHide);

	p_tyC0009Info ACCESS ADR(tyCommon.tyInfo);

	p_tyP1030MagSet ACCESS ADR(tyP1030MagSet.tyMagSet);

	IF bTeachTravPosMag1 OR bTeachTravPosMag2 OR bTeachTravPosMag3 OR bTeachTravPosMag4
		OR bTeachLifterMag1Slt1Pos OR bTeachLifterMag2Slt1Pos OR bTeachLifterMag3Slt1Pos OR bTeachLifterMag4Slt1Pos THEN
		bTeachTravPosMag1		:= FALSE;
		bTeachTravPosMag2		:= FALSE;
		bTeachTravPosMag3		:= FALSE;
		bTeachTravPosMag4		:= FALSE;
		bTeachLifterMag1Slt1Pos	:= FALSE;
		bTeachLifterMag2Slt1Pos	:= FALSE;
		bTeachLifterMag3Slt1Pos	:= FALSE;
		bTeachLifterMag4Slt1Pos	:= FALSE;
		bTeachServo				:= FALSE;
	ELSE
		udiP1030SelectedRowOld	 := 0;
	END_IF

	// Enabling Auto Detect Magazine Model Setting
	tyP1030MagSet.tyMagSet.tyDrpDnMagModel.uiRtStat := NOT(p_tyNtParamCurr.bMagAutoVerifyPrep);
	tyP1030MagSet.tyMagSet.tyTxtMagModel.uiRtStat	:= NOT(p_tyNtParamCurr.bMagAutoVerifyPrep);

END_ACTION
```

#### Act_OptP1030Del.st
```iecst
ACTION Act_OptP1030Del:

	CASE p_tyNtParamCurr.eProjMag OF
		LDMagDual, LDMagTriple:

			IF tyP1030MagSet.tyMagSet.tyBtnDelete.bRtCompl = TRUE THEN
				IF usiDelMagRcpStep = 0 THEN
					tyP1030MagSet.tyMagSet.tyTableRecipe.uiMaskRtStat					:= FALSE;

					IF tyP1030MagSet.tyMagSet.tyTableRecipe.a_tyStringDataCol1[tyP1030Table.uiSelectedRow].sValue = p_tyMagRcpCurrRcp.sRcpNm THEN
						p_tyC0008MsgBox ACCESS ADR(tyP1030MagSet.tyMsgBoxDelCurrRcpAsk);

						IF tyP1030MagSet.tyMsgBoxDelCurrRcpAsk.tyBtnNo.bRtCompl = TRUE THEN
							tyP1030MagSet.tyMsgBoxDelCurrRcpAsk.tyBtnNo.bRtCompl 	:= FALSE;
							tyP1030MagSet.tyMsgBoxDelCurrRcpAsk.tyBtnNo.bValue 		:= FALSE;

							p_tyC0008MsgBox ACCESS ADR(tyP1030MagSet.tyMsgBoxHide);

							usiDelMagRcpStep	:= 99;
						END_IF
					ELSE
						p_tyC0008MsgBox ACCESS ADR(tyP1030MagSet.tyMsgBoxDelAsk);

						IF tyP1030MagSet.tyMsgBoxDelAsk.tyBtnYes.bRtCompl = TRUE THEN
							tyP1030MagSet.tyMsgBoxDelAsk.tyBtnYes.bRtCompl				:= FALSE;
							tyP1030MagSet.tyMsgBoxDelAsk.tyBtnYes.bValue				:= FALSE;

							p_tyC0008MsgBox ACCESS ADR(tyP1030MagSet.tyMsgBoxHide);

							usiDelMagRcpStep	:= 1;

						ELSIF tyP1030MagSet.tyMsgBoxDelAsk.tyBtnNo.bRtCompl = TRUE THEN
							tyP1030MagSet.tyMsgBoxDelAsk.tyBtnNo.bRtCompl			:= FALSE;
							tyP1030MagSet.tyMsgBoxDelAsk.tyBtnNo.bValue				:= FALSE;

							p_tyC0008MsgBox ACCESS ADR(tyP1030MagSet.tyMsgBoxHide);

							usiDelMagRcpStep	:= 99;

						END_IF
					END_IF

				ELSIF usiDelMagRcpStep = 1 THEN
					tyMagRcpInfoIn.sRcpNm			:= tyP1030MagSet.tyMagSet.tyTableRecipe.a_tyStringDataCol1[tyP1030Table.uiSelectedRow].sValue;

					eMagRcpAct					:= MagRcpActDel;

					IF p_eMagRcpStat = MagRcpActDel AND p_eMagRcpStatus = Done THEN
						eMagRcpAct				:= MagRcpActIdle;

						IF p_bMagRcpNmEmpty = TRUE THEN
							usiDelMagRcpStep		:= 2;
						ELSIF p_bMagRcpNmNotExist = TRUE THEN
							usiDelMagRcpStep		:= 3;
						ELSE
							bRefreshMagRcpTable		:= TRUE;
							bRefreshMagRcpDetail	:= TRUE;
							usiDelMagRcpStep		:= 99;
						END_IF

					ELSIF p_eMagRcpStatus = Error THEN
						p_tyC0008MsgBox ACCESS ADR(tyP1030MagSet.tyMsgBoxDelErr);

						IF tyP1030MagSet.tyMsgBoxDelErr.tyBtnNo.bRtCompl = TRUE THEN
							tyP1030MagSet.tyMsgBoxDelErr.tyBtnNo.bRtCompl 				:= FALSE;
							tyP1030MagSet.tyMsgBoxDelErr.tyBtnNo.bValue 				:= FALSE;

							p_tyC0008MsgBox ACCESS ADR(tyP1030MagSet.tyMsgBoxHide);

							usiDelMagRcpStep		:= 99;
						END_IF
					END_IF

				ELSIF usiDelMagRcpStep = 2 THEN
					p_tyC0008MsgBox ACCESS ADR(tyP1030MagSet.tyMsgBoxDelNmEmpty);

					IF tyP1030MagSet.tyMsgBoxDelNmEmpty.tyBtnNo.bRtCompl = TRUE THEN
						tyP1030MagSet.tyMsgBoxDelNmEmpty.tyBtnNo.bRtCompl 				:= FALSE;
						tyP1030MagSet.tyMsgBoxDelNmEmpty.tyBtnNo.bValue 				:= FALSE;

						p_tyC0008MsgBox ACCESS ADR(tyP1030MagSet.tyMsgBoxHide);

						usiDelMagRcpStep		:= 99;
					END_IF

				ELSIF usiDelMagRcpStep = 3 THEN
					p_tyC0008MsgBox ACCESS ADR(tyP1030MagSet.tyMsgBoxDelNmNotExist);

					IF tyP1030MagSet.tyMsgBoxDelNmNotExist.tyBtnNo.bRtCompl = TRUE THEN
						tyP1030MagSet.tyMsgBoxDelNmNotExist.tyBtnNo.bRtCompl 	:= FALSE;
						tyP1030MagSet.tyMsgBoxDelNmNotExist.tyBtnNo.bValue 		:= FALSE;

						p_tyC0008MsgBox ACCESS ADR(tyP1030MagSet.tyMsgBoxHide);

						usiDelMagRcpStep	:= 99;
					END_IF

				ELSIF usiDelMagRcpStep = 99 THEN
					bRefreshMagRcpTable	:= FALSE;

					//Unmask
					tyP1030MagSet.tyMagSet.tyTableRecipe.uiMaskRtStat			:= TRUE;

					//Reset
					tyP1030MagSet.tyMagSet.tyBtnDelete.bRtCompl					:= FALSE;
					tyP1030MagSet.tyMagSet.tyBtnDelete.bValue					:= FALSE;

					usiDelMagRcpStep		:= 0;
				END_IF

			END_IF

		LDMagQuadruple:
			IF tyP1030MagSet.tyMagSet.tyBtnDelete.bRtCompl = TRUE THEN
				IF usiDelMagRcpStep = 0 THEN
					tyP1030MagSet.tyMagSet.tyTableRecipe.uiMaskRtStat					:= FALSE;

					IF tyP1030MagSet.tyMagSet.tyTableRecipe.a_tyStringDataCol1[tyP1030Table.uiSelectedRow].sValue = p_tyMagRcpCurrRcp.sRcpNm THEN
						p_tyC0008MsgBox ACCESS ADR(tyP1030MagSet.tyMsgBoxDelCurrRcpAsk);

						IF tyP1030MagSet.tyMsgBoxDelCurrRcpAsk.tyBtnNo.bRtCompl = TRUE THEN
							tyP1030MagSet.tyMsgBoxDelCurrRcpAsk.tyBtnNo.bRtCompl 	:= FALSE;
							tyP1030MagSet.tyMsgBoxDelCurrRcpAsk.tyBtnNo.bValue 		:= FALSE;

							p_tyC0008MsgBox ACCESS ADR(tyP1030MagSet.tyMsgBoxHide);

							usiDelMagRcpStep	:= 99;
						END_IF
					ELSE
						p_tyC0008MsgBox ACCESS ADR(tyP1030MagSet.tyMsgBoxDelAsk);

						IF tyP1030MagSet.tyMsgBoxDelAsk.tyBtnYes.bRtCompl = TRUE THEN
							tyP1030MagSet.tyMsgBoxDelAsk.tyBtnYes.bRtCompl				:= FALSE;
							tyP1030MagSet.tyMsgBoxDelAsk.tyBtnYes.bValue				:= FALSE;

							p_tyC0008MsgBox ACCESS ADR(tyP1030MagSet.tyMsgBoxHide);

							usiDelMagRcpStep	:= 1;

						ELSIF tyP1030MagSet.tyMsgBoxDelAsk.tyBtnNo.bRtCompl = TRUE THEN
							tyP1030MagSet.tyMsgBoxDelAsk.tyBtnNo.bRtCompl			:= FALSE;
							tyP1030MagSet.tyMsgBoxDelAsk.tyBtnNo.bValue				:= FALSE;

							p_tyC0008MsgBox ACCESS ADR(tyP1030MagSet.tyMsgBoxHide);

							usiDelMagRcpStep	:= 99;

						END_IF
					END_IF

				ELSIF usiDelMagRcpStep = 1 THEN
					tyMagRcpInfoIn.sRcpNm			:= tyP1030MagSet.tyMagSet.tyTableRecipe.a_tyStringDataCol1[tyP1030Table.uiSelectedRow].sValue;
					tyMagRcpInfoIn1.sRcpNm			:= tyP1030MagSet.tyMagSet.tyTableRecipe.a_tyStringDataCol1[tyP1030Table.uiSelectedRow].sValue;
					eMagRcpAct					:= MagRcpActDel;
					eMagRcpAct1					:= MagRcpActDel;
					IF (p_eMagRcpStat = MagRcpActDel AND p_eMagRcpStatus = Done)
						AND (p_eMagRcpStat1 = MagRcpActDel AND p_eMagRcpStatus1 = Done)
						THEN
						eMagRcpAct				:= MagRcpActIdle;

						IF p_bMagRcpNmEmpty = TRUE OR p_bMagRcpNmEmpty1 = TRUE THEN
							usiDelMagRcpStep		:= 2;
						ELSIF p_bMagRcpNmNotExist = TRUE OR p_bMagRcpNmNotExist1 = TRUE THEN
							usiDelMagRcpStep		:= 3;
						ELSE
							bRefreshMagRcpTable		:= TRUE;
							bRefreshMagRcpDetail	:= TRUE;
							usiDelMagRcpStep		:= 99;
						END_IF

					ELSIF p_eMagRcpStatus = Error OR p_eMagRcpStatus1 = Error THEN
						p_tyC0008MsgBox ACCESS ADR(tyP1030MagSet.tyMsgBoxDelErr);

						IF tyP1030MagSet.tyMsgBoxDelErr.tyBtnNo.bRtCompl = TRUE THEN
							tyP1030MagSet.tyMsgBoxDelErr.tyBtnNo.bRtCompl 				:= FALSE;
							tyP1030MagSet.tyMsgBoxDelErr.tyBtnNo.bValue 				:= FALSE;

							p_tyC0008MsgBox ACCESS ADR(tyP1030MagSet.tyMsgBoxHide);

							usiDelMagRcpStep		:= 99;
						END_IF
					END_IF

				ELSIF usiDelMagRcpStep = 2 THEN
					p_tyC0008MsgBox ACCESS ADR(tyP1030MagSet.tyMsgBoxDelNmEmpty);

					IF tyP1030MagSet.tyMsgBoxDelNmEmpty.tyBtnNo.bRtCompl = TRUE THEN
						tyP1030MagSet.tyMsgBoxDelNmEmpty.tyBtnNo.bRtCompl 				:= FALSE;
						tyP1030MagSet.tyMsgBoxDelNmEmpty.tyBtnNo.bValue 				:= FALSE;

						p_tyC0008MsgBox ACCESS ADR(tyP1030MagSet.tyMsgBoxHide);

						usiDelMagRcpStep		:= 99;
					END_IF

				ELSIF usiDelMagRcpStep = 3 THEN
					p_tyC0008MsgBox ACCESS ADR(tyP1030MagSet.tyMsgBoxDelNmNotExist);

					IF tyP1030MagSet.tyMsgBoxDelNmNotExist.tyBtnNo.bRtCompl = TRUE THEN
						tyP1030MagSet.tyMsgBoxDelNmNotExist.tyBtnNo.bRtCompl 	:= FALSE;
						tyP1030MagSet.tyMsgBoxDelNmNotExist.tyBtnNo.bValue 		:= FALSE;

						p_tyC0008MsgBox ACCESS ADR(tyP1030MagSet.tyMsgBoxHide);

						usiDelMagRcpStep	:= 99;
					END_IF

				ELSIF usiDelMagRcpStep = 99 THEN
					bRefreshMagRcpTable	:= FALSE;

					//Unmask
					tyP1030MagSet.tyMagSet.tyTableRecipe.uiMaskRtStat			:= TRUE;

					//Reset
					tyP1030MagSet.tyMagSet.tyBtnDelete.bRtCompl					:= FALSE;
					tyP1030MagSet.tyMagSet.tyBtnDelete.bValue					:= FALSE;

					usiDelMagRcpStep		:= 0;
				END_IF

			END_IF
		END_CASE
END_ACTION
```

#### Act_OptP1030Keypad.st
```iecst
ACTION Act_OptP1030Keypad:

	IF fUIOutRtStatTPIsOpen(ADR(tyP1030MagSet.tyMagSet.tyStringRecipeNm.uiRtStat)) THEN
		tyProperty.tyKeypad.tyStringTitle.sKeypadTitle	:= tyP1030MagSet.tyMagSet.tyStringRecipeNm.sKeypadTitle;

	ELSIF fUIOutRtStatTPIsOpen(ADR(tyP1030MagSet.tyMagSet.tyNumSltToSltDist.uiRtStat)) THEN
		tyProperty.tyKeypad.tyStringTitle.sKeypadTitle	:= tyP1030MagSet.tyMagSet.tyNumSltToSltDist.sKeypadTitle;

	ELSIF fUIOutRtStatTPIsOpen(ADR(tyP1030MagSet.tyMagSet.tyNumMaxSlt.uiRtStat)) THEN
		tyProperty.tyKeypad.tyStringTitle.sKeypadTitle	:= tyP1030MagSet.tyMagSet.tyNumMaxSlt.sKeypadTitle;

	ELSIF fUIOutRtStatTPIsOpen(ADR(tyP1030MagSet.tyMagSet.tyNumLifterMag1Slt1Pos.uiRtStat)) THEN
		tyProperty.tyKeypad.tyStringTitle.sKeypadTitle	:= tyP1030MagSet.tyMagSet.tyNumLifterMag1Slt1Pos.sKeypadTitle;

	ELSIF fUIOutRtStatTPIsOpen(ADR(tyP1030MagSet.tyMagSet.tyNumLifterMag2Slt1Pos.uiRtStat)) THEN
		tyProperty.tyKeypad.tyStringTitle.sKeypadTitle	:= tyP1030MagSet.tyMagSet.tyNumLifterMag2Slt1Pos.sKeypadTitle;

	ELSIF fUIOutRtStatTPIsOpen(ADR(tyP1030MagSet.tyMagSet.tyNumLifterMag3Slt1Pos.uiRtStat)) THEN
		tyProperty.tyKeypad.tyStringTitle.sKeypadTitle	:= tyP1030MagSet.tyMagSet.tyNumLifterMag3Slt1Pos.sKeypadTitle;

	ELSIF fUIOutRtStatTPIsOpen(ADR(tyP1030MagSet.tyMagSet.tyNumLifterMag4Slt1Pos.uiRtStat)) THEN
		tyProperty.tyKeypad.tyStringTitle.sKeypadTitle	:= tyP1030MagSet.tyMagSet.tyNumLifterMag4Slt1Pos.sKeypadTitle;

	ELSIF fUIOutRtStatTPIsOpen(ADR(tyP1030MagSet.tyMagSet.tyNumTravPosMag1.uiRtStat)) THEN
		tyProperty.tyKeypad.tyStringTitle.sKeypadTitle	:= tyP1030MagSet.tyMagSet.tyNumTravPosMag1.sKeypadTitle;

	ELSIF fUIOutRtStatTPIsOpen(ADR(tyP1030MagSet.tyMagSet.tyNumTravPosMag2.uiRtStat)) THEN
		tyProperty.tyKeypad.tyStringTitle.sKeypadTitle	:= tyP1030MagSet.tyMagSet.tyNumTravPosMag2.sKeypadTitle;

	ELSIF fUIOutRtStatTPIsOpen(ADR(tyP1030MagSet.tyMagSet.tyNumTravPosMag3.uiRtStat)) THEN
		tyProperty.tyKeypad.tyStringTitle.sKeypadTitle	:= tyP1030MagSet.tyMagSet.tyNumTravPosMag3.sKeypadTitle;

	ELSIF fUIOutRtStatTPIsOpen(ADR(tyP1030MagSet.tyMagSet.tyNumTravPosMag4.uiRtStat)) THEN
		tyProperty.tyKeypad.tyStringTitle.sKeypadTitle	:= tyP1030MagSet.tyMagSet.tyNumTravPosMag3.sKeypadTitle;

	ELSIF fUIOutRtStatTPIsOpen(ADR(tyP1030MagSet.tyMagSet.tyNumMagMaxBrdWidth.uiRtStat)) THEN
		tyProperty.tyKeypad.tyStringTitle.sKeypadTitle  := tyP1030MagSet.tyMagSet.tyNumMagMaxBrdWidth.sKeypadTitle;
	ELSE
		tyProperty.tyKeypad.tyStringTitle.sKeypadTitle	:= '';

	END_IF

END_ACTION
```

#### Act_OptP1030LoadData.st
```iecst
ACTION Act_OptP1030LoadData:

	udiP1030SelectedRow		:= STRING_TO_UDINT(tyP1030MagSet.tyMagSet.tyTableRecipe.a_tyStringDataCol0[tyP1030Table.uiSelectedRow].sValue);

	IF udiP1030SelectedRow <> udiP1030SelectedRowOld OR bRefreshMagRcpDetail = TRUE OR bUpdateP1030LoadData THEN

		IF tyP1030MagSet.tyMagSet.tyTableRecipe.a_tyStringDataCol1[tyP1030Table.uiSelectedRow].sValue <> '' THEN
			//Update Recipe Data
			IF tyP1030MagSet.tyMagSet.tyBtnSort.bValue THEN
				tyP1030MagSet.tyMagSet.tyStringRecipeNm.sValue			:= p_tyMagRcpSortedList[udiP1030SelectedRow].sRcpNm;
				tyP1030MagSet.tyMagSet.tyNumSltToSltDist.diValue		:= p_tyMagRcpSortedList[udiP1030SelectedRow].diSltToSltInUM;
				tyP1030MagSet.tyMagSet.tyNumMaxSlt.diValue				:= p_tyMagRcpSortedList[udiP1030SelectedRow].diTtlSlt;
				tyP1030MagSet.tyMagSet.tyNumLifterMag1Slt1Pos.diValue	:= p_tyMagRcpSortedList[udiP1030SelectedRow].diMag1Slt1PosInUM;
				tyP1030MagSet.tyMagSet.tyNumLifterMag2Slt1Pos.diValue	:= p_tyMagRcpSortedList[udiP1030SelectedRow].diMag2Slt1PosInUM;
				tyP1030MagSet.tyMagSet.tyNumLifterMag3Slt1Pos.diValue	:= p_tyMagRcpSortedList[udiP1030SelectedRow].diMag3Slt1PosInUM;
				tyP1030MagSet.tyMagSet.tyNumLifterMag4Slt1Pos.diValue	:= p_tyMagRcpSortedList[udiP1030SelectedRow].diMag4Slt1PosInUM;
				tyP1030MagSet.tyMagSet.tyNumTravPosMag1.diValue			:= p_tyMagRcpSortedList[udiP1030SelectedRow].diMag1TravPosInUM;
				tyP1030MagSet.tyMagSet.tyNumTravPosMag2.diValue			:= p_tyMagRcpSortedList[udiP1030SelectedRow].diMag2TravPosInUM;
				tyP1030MagSet.tyMagSet.tyNumTravPosMag3.diValue			:= p_tyMagRcpSortedList[udiP1030SelectedRow].diMag3TravPosInUM;
				tyP1030MagSet.tyMagSet.tyNumTravPosMag4.diValue			:= p_tyMagRcpSortedList[udiP1030SelectedRow].diMag4TravPosInUM;
				tyP1030MagSet.tyMagSet.tyDrpDnMagModel.usiValueIdx		:= p_tyMagRcpSortedList[udiP1030SelectedRow].usiMagModel;
				tyP1030MagSet.tyMagSet.tyNumMagMaxBrdWidth.diValue		:= p_tyMagRcpSortedList[udiP1030SelectedRow].diMagMaxBrdWidth;
				tyP1030MagSet.tyMagSet.tyBtnSafetyBarDisabled.bValue	:= p_tyMagRcpSortedList[udiP1030SelectedRow].bSafetyBarDisabled;
				tyP1030MagSet.tyMagSet.tyBtnMagHeightChkEn.bValue		:= p_tyMagRcpSortedList[udiP1030SelectedRow].bMagHeightChkEn;
			ELSE
				tyP1030MagSet.tyMagSet.tyStringRecipeNm.sValue			:= p_tyMagRcpCurrList[udiP1030SelectedRow].sRcpNm;
				tyP1030MagSet.tyMagSet.tyNumSltToSltDist.diValue		:= p_tyMagRcpCurrList[udiP1030SelectedRow].diSltToSltInUM;
				tyP1030MagSet.tyMagSet.tyNumMaxSlt.diValue				:= p_tyMagRcpCurrList[udiP1030SelectedRow].diTtlSlt;
				tyP1030MagSet.tyMagSet.tyNumLifterMag1Slt1Pos.diValue	:= p_tyMagRcpCurrList[udiP1030SelectedRow].diMag1Slt1PosInUM;
				tyP1030MagSet.tyMagSet.tyNumLifterMag2Slt1Pos.diValue	:= p_tyMagRcpCurrList[udiP1030SelectedRow].diMag2Slt1PosInUM;
				tyP1030MagSet.tyMagSet.tyNumLifterMag3Slt1Pos.diValue	:= p_tyMagRcpCurrList[udiP1030SelectedRow].diMag3Slt1PosInUM;
				tyP1030MagSet.tyMagSet.tyNumLifterMag4Slt1Pos.diValue	:= p_tyMagRcpCurrList[udiP1030SelectedRow].diMag4Slt1PosInUM;
				tyP1030MagSet.tyMagSet.tyNumTravPosMag1.diValue			:= p_tyMagRcpCurrList[udiP1030SelectedRow].diMag1TravPosInUM;
				tyP1030MagSet.tyMagSet.tyNumTravPosMag2.diValue			:= p_tyMagRcpCurrList[udiP1030SelectedRow].diMag2TravPosInUM;
				tyP1030MagSet.tyMagSet.tyNumTravPosMag3.diValue			:= p_tyMagRcpCurrList[udiP1030SelectedRow].diMag3TravPosInUM;
				tyP1030MagSet.tyMagSet.tyNumTravPosMag4.diValue			:= p_tyMagRcpCurrList[udiP1030SelectedRow].diMag4TravPosInUM;
				tyP1030MagSet.tyMagSet.tyDrpDnMagModel.usiValueIdx		:= p_tyMagRcpCurrList[udiP1030SelectedRow].usiMagModel;
				tyP1030MagSet.tyMagSet.tyNumMagMaxBrdWidth.diValue		:= p_tyMagRcpCurrList[udiP1030SelectedRow].diMagMaxBrdWidth;
				tyP1030MagSet.tyMagSet.tyBtnSafetyBarDisabled.bValue	:= p_tyMagRcpCurrList[udiP1030SelectedRow].bSafetyBarDisabled;
				tyP1030MagSet.tyMagSet.tyBtnMagHeightChkEn.bValue		:= p_tyMagRcpCurrList[udiP1030SelectedRow].bMagHeightChkEn;
			END_IF
		ELSE

			tyP1030MagSet.tyMagSet.tyStringRecipeNm.sValue			:= '';
			tyP1030MagSet.tyMagSet.tyNumSltToSltDist.diValue		:= 10000;
			tyP1030MagSet.tyMagSet.tyNumMaxSlt.diValue				:= p_tyNtParamCurr.diProjMagMaxSlt;
			tyP1030MagSet.tyMagSet.tyNumLifterMag1Slt1Pos.diValue	:= 0;
			tyP1030MagSet.tyMagSet.tyNumLifterMag2Slt1Pos.diValue	:= 0;
			tyP1030MagSet.tyMagSet.tyNumLifterMag3Slt1Pos.diValue	:= 0;
			tyP1030MagSet.tyMagSet.tyNumLifterMag4Slt1Pos.diValue	:= 0;
			tyP1030MagSet.tyMagSet.tyNumTravPosMag1.diValue			:= 0;
			tyP1030MagSet.tyMagSet.tyNumTravPosMag2.diValue			:= 0;
			tyP1030MagSet.tyMagSet.tyNumTravPosMag3.diValue			:= 0;
			tyP1030MagSet.tyMagSet.tyNumTravPosMag4.diValue			:= 0;
			tyP1030MagSet.tyMagSet.tyDrpDnMagModel.usiValueIdx		:= 0;
			tyP1030MagSet.tyMagSet.tyNumMagMaxBrdWidth.diValue		:= 0;
			tyP1030MagSet.tyMagSet.tyBtnSafetyBarDisabled.bValue	:= FALSE;
			tyP1030MagSet.tyMagSet.tyBtnMagHeightChkEn.bValue		:= FALSE;
		END_IF

		bRefreshMagRcpDetail	:= FALSE;
		bUpdateP1030LoadData	:= FALSE;
		udiP1030SelectedRowOld 	:= udiP1030SelectedRow;

		fUIInRtStatOff(ADR(tyP1030MagSet.tyMagSet.tyBtnSave.uiMaskRtStat));

	END_IF

END_ACTION
```

#### Act_OptP1030Mask.st
```iecst
ACTION Act_OptP1030Mask:

	IF tyP1030MagSet.tyMagSet.tyStringRecipeNm.bRtCompl				OR tyP1030MagSet.tyMagSet.tyNumSltToSltDist.bRtCompl
		OR tyP1030MagSet.tyMagSet.tyNumMaxSlt.bRtCompl				OR tyP1030MagSet.tyMagSet.tyNumLifterMag1Slt1Pos.bRtCompl
		OR tyP1030MagSet.tyMagSet.tyNumLifterMag2Slt1Pos.bRtCompl	OR tyP1030MagSet.tyMagSet.tyNumLifterMag3Slt1Pos.bRtCompl
		OR tyP1030MagSet.tyMagSet.tyNumLifterMag4Slt1Pos.bRtCompl
		OR tyP1030MagSet.tyMagSet.tyNumTravPosMag1.bRtCompl			OR tyP1030MagSet.tyMagSet.tyNumTravPosMag2.bRtCompl
		OR tyP1030MagSet.tyMagSet.tyNumTravPosMag3.bRtCompl			OR tyP1030MagSet.tyMagSet.tyNumTravPosMag4.bRtCompl
		OR tyP1030MagSet.tyMagSet.tyDrpDnMagModel.bRtCompl			OR tyP1030MagSet.tyMagSet.tyNumMagMaxBrdWidth.bRtCompl
		OR tyP1030MagSet.tyMagSet.tyBtnSafetyBarDisabled.bRtCompl 	OR tyP1030MagSet.tyMagSet.tyBtnMagHeightChkEn.bRtCompl
		THEN

		fUIInRtStatHide(ADR(tyP1030MagSet.tyMagSet.tyBtnSave.uiMaskRtStat));

		tyP1030MagSet.tyMagSet.tyStringRecipeNm.bRtCompl		:= FALSE;
		tyP1030MagSet.tyMagSet.tyNumSltToSltDist.bRtCompl		:= FALSE;
		tyP1030MagSet.tyMagSet.tyNumMaxSlt.bRtCompl				:= FALSE;
		tyP1030MagSet.tyMagSet.tyNumLifterMag1Slt1Pos.bRtCompl	:= FALSE;
		tyP1030MagSet.tyMagSet.tyNumLifterMag2Slt1Pos.bRtCompl	:= FALSE;
		tyP1030MagSet.tyMagSet.tyNumLifterMag3Slt1Pos.bRtCompl	:= FALSE;
		tyP1030MagSet.tyMagSet.tyNumLifterMag4Slt1Pos.bRtCompl	:= FALSE;
		tyP1030MagSet.tyMagSet.tyNumTravPosMag1.bRtCompl		:= FALSE;
		tyP1030MagSet.tyMagSet.tyNumTravPosMag2.bRtCompl		:= FALSE;
		tyP1030MagSet.tyMagSet.tyNumTravPosMag3.bRtCompl		:= FALSE;
		tyP1030MagSet.tyMagSet.tyNumTravPosMag4.bRtCompl		:= FALSE;
		tyP1030MagSet.tyMagSet.tyDrpDnMagModel.bRtCompl			:= FALSE;
		tyP1030MagSet.tyMagSet.tyNumMagMaxBrdWidth.bRtCompl		:= FALSE;
		tyP1030MagSet.tyMagSet.tyBtnSafetyBarDisabled.bRtCompl	:= FALSE;
		tyP1030MagSet.tyMagSet.tyBtnMagHeightChkEn.bRtCompl		:= FALSE;
	END_IF

	IF tyP1030MagSet.tyMagSet.tyTableRecipe.a_tyStringDataCol1[tyP1030Table.uiSelectedRow].sValue <> '' THEN
		fUIInRtStatHide(ADR(tyP1030MagSet.tyMagSet.tyBtnDelete.uiMaskRtStat));
	ELSE
		fUIInRtStatOff(ADR(tyP1030MagSet.tyMagSet.tyBtnDelete.uiMaskRtStat));
	END_IF

	tyP1030MagSet.tyMagSet.tyBtnSort.uiMaskRtStat.0		:= (tyP1030MagSet.tyMagSet.tyTableRecipe.a_tyStringDataCol1[1].sValue <> '')
	AND (tyP1030MagSet.tyMagSet.tyBtnSave.uiMaskRtStat.0 = FALSE) AND (tyP1030MagSet.tyMagSet.tyBtnDelete.bRtCompl = FALSE) ;

END_ACTION
```
